LIN {X 0,Y 310.928,Z 762.241,A -85,B 0,C 180,E1 -15746.111,E2 -15746.111} C_VEL
LIN {X 0,Y 310.701,Z 763.849,A -85,B 0,C 180,E1 -15748.703,E2 -15748.703} C_VEL
LIN {X 0,Y 310.698,Z 764.081,A -85,B 0,C 180,E1 -15749.999,E2 -15749.999} C_VEL
LIN {X 0,Y 310.7,Z 763.891,A -85,B 0,C 180,E1 -15751.295,E2 -15751.295} C_VEL
LIN {X 0,Y 310.923,Z 762.339,A -85,B 0,C 180,E1 -15753.887,E2 -15753.887} C_VEL
LIN {X 0,Y 311.084,Z 760.984,A -85,B 0,C 180,E1 -15755.184,E2 -15755.184} C_VEL
LIN {X 0,Y 311.392,Z 758.118,A -85,B 0,C 180,E1 -15757.129,E2 -15757.129} C_VEL
LIN {X 0,Y 311.868,Z 754.229,A -85,B 0,C 180,E1 -15759.075,E2 -15759.075} C_VEL
LIN {X 0,Y 312.703,Z 749.212,A -85,B 0,C 180,E1 -15761.012,E2 -15761.012} C_VEL
LIN {X 0,Y 313.678,Z 742.897,A -85,B 0,C 180,E1 -15762.946,E2 -15762.946} C_VEL
LIN {X 0,Y 314.945,Z 734.989,A -85,B 0,C 180,E1 -15764.868,E2 -15764.868} C_VEL
LIN {X 0,Y 316.624,Z 725.146,A -85,B 0,C 180,E1 -15766.77,E2 -15766.77} C_VEL
LIN {X 0,Y 317.967,Z 714.82,A -85,B 0,C 180,E1 -15768.357,E2 -15768.357} C_VEL
LIN {X 0,Y 319.245,Z 704.591,A -85,B 0,C 180,E1 -15769.615,E2 -15769.615} C_VEL
LIN {X 0,Y 320.576,Z 693.385,A -85,B 0,C 180,E1 -15770.701,E2 -15770.701} C_VEL
LIN {X 0,Y 321.765,Z 680.745,A -85,B 0,C 180,E1 -15771.627,E2 -15771.627} C_VEL
LIN {X 0,Y 322.52,Z 668.996,A -85,B 0,C 180,E1 -15772.247,E2 -15772.247} C_VEL
LIN {X 0,Y 323.102,Z 656.548,A -85,B 0,C 180,E1 -15772.668,E2 -15772.668} C_VEL
LIN {X 0,Y 324.626,Z 584.757,A -85,B 0,C 180,E1 -15774.261,E2 -15774.261} C_VEL
LIN {X 0,Y 322.955,Z 579.324,A -85,B 0,C 180,E1 -15774.526,E2 -15774.526} C_VEL
LIN {X 0,Y 320.223,Z 574.422,A -85,B 0,C 180,E1 -15774.87,E2 -15774.87} C_VEL
LIN {X 0,Y 311.253,Z 562.348,A -85,B 0,C 180,E1 -15775.948,E2 -15775.948} C_VEL
LIN {X 0,Y 309.308,Z 559.08,A -85,B 0,C 180,E1 -15776.208,E2 -15776.208} C_VEL
LIN {X 0,Y 307.194,Z 553.881,A -85,B 0,C 180,E1 -15776.597,E2 -15776.597} C_VEL
LIN {X 0,Y 305.556,Z 546.682,A -85,B 0,C 180,E1 -15779.186,E2 -15779.186} C_VEL
LIN {X 0,Y 305.497,Z 546.411,A -85,B 0,C 180,E1 -15779.66,E2 -15779.66} C_VEL
LIN {X 0,Y 305.462,Z 546.438,A -85,B 0,C 180,E1 -15784.077,E2 -15784.077} C_VEL
LIN {X 0,Y 305.499,Z 546.425,A -85,B 0,C 180,E1 -15786.734,E2 -15786.734} C_VEL
LIN {X 0,Y 305.452,Z 546.427,A -85,B 0,C 180,E1 -15790.599,E2 -15790.599} C_VEL
LIN {X 0,Y 305.423,Z 546.43,A -85,B 0,C 180,E1 -15793.654,E2 -15793.654} C_VEL
LIN {X 0,Y 305.482,Z 546.432,A -85,B 0,C 180,E1 -15797.407,E2 -15797.407} C_VEL
LIN {X 0,Y 305.504,Z 546.404,A -85,B 0,C 180,E1 -15801.601,E2 -15801.601} C_VEL
LIN {X 0,Y 305.458,Z 546.435,A -85,B 0,C 180,E1 -15804.886,E2 -15804.886} C_VEL
LIN {X 0,Y 305.447,Z 546.433,A -85,B 0,C 180,E1 -15808.354,E2 -15808.354} C_VEL
LIN {X 0,Y 305.515,Z 546.426,A -85,B 0,C 180,E1 -15811.113,E2 -15811.113} C_VEL
LIN {X 0,Y 305.565,Z 546.421,A -85,B 0,C 180,E1 -15814.087,E2 -15814.087} C_VEL
LIN {X 0,Y 305.494,Z 546.421,A -85,B 0,C 180,E1 -15818.402,E2 -15818.402} C_VEL
LIN {X 0,Y 305.583,Z 546.42,A -85,B 0,C 180,E1 -15821.217,E2 -15821.217} C_VEL
LIN {X 0,Y 305.642,Z 546.405,A -85,B 0,C 180,E1 -15825.349,E2 -15825.349} C_VEL
LIN {X 0,Y 305.631,Z 546.402,A -85,B 0,C 180,E1 -15829.399,E2 -15829.399} C_VEL
LIN {X 0,Y 305.806,Z 546.391,A -85,B 0,C 180,E1 -15832.074,E2 -15832.074} C_VEL
LIN {X 0,Y 305.683,Z 546.405,A -85,B 0,C 180,E1 -15834.723,E2 -15834.723} C_VEL
LIN {X 0,Y 305.952,Z 546.368,A -85,B 0,C 180,E1 -15838.684,E2 -15838.684} C_VEL
LIN {X 0,Y 305.952,Z 546.374,A -85,B 0,C 180,E1 -15841.316,E2 -15841.316} C_VEL
LIN {X 0,Y 305.847,Z 546.385,A -85,B 0,C 180,E1 -15846.597,E2 -15846.597} C_VEL
LIN {X 0,Y 305.729,Z 546.392,A -85,B 0,C 180,E1 -15849.26,E2 -15849.26} C_VEL
LIN {X 0,Y 305.584,Z 546.42,A -85,B 0,C 180,E1 -15853.296,E2 -15853.296} C_VEL
LIN {X 0,Y 305.587,Z 546.407,A -85,B 0,C 180,E1 -15856.02,E2 -15856.02} C_VEL
LIN {X 0,Y 305.574,Z 546.424,A -85,B 0,C 180,E1 -15859.448,E2 -15859.448} C_VEL
LIN {X 0,Y 305.484,Z 546.427,A -85,B 0,C 180,E1 -15863.042,E2 -15863.042} C_VEL
LIN {X 0,Y 305.519,Z 546.418,A -85,B 0,C 180,E1 -15866.219,E2 -15866.219} C_VEL
LIN {X 0,Y 305.482,Z 546.433,A -85,B 0,C 180,E1 -15869.048,E2 -15869.048} C_VEL
LIN {X 0,Y 305.436,Z 546.436,A -85,B 0,C 180,E1 -15871.953,E2 -15871.953} C_VEL
LIN {X 0,Y 305.457,Z 546.422,A -85,B 0,C 180,E1 -15875.114,E2 -15875.114} C_VEL
LIN {X 0,Y 305.444,Z 546.433,A -85,B 0,C 180,E1 -15878.53,E2 -15878.53} C_VEL
LIN {X 0,Y 305.48,Z 546.416,A -85,B 0,C 180,E1 -15882.593,E2 -15882.593} C_VEL
LIN {X 0,Y 305.488,Z 546.423,A -85,B 0,C 180,E1 -15886.358,E2 -15886.358} C_VEL
LIN {X 0,Y 305.495,Z 546.425,A -85,B 0,C 180,E1 -15889.9,E2 -15889.9} C_VEL
LIN {X 0,Y 305.497,Z 546.41,A -85,B 0,C 180,E1 -15893.628,E2 -15893.628} C_VEL
LIN {X 0,Y 305.507,Z 546.515,A -85,B 0,C 180,E1 -15896.35,E2 -15896.35} C_VEL
LIN {X 0,Y 307.874,Z 556.829,A -85,B 0,C 180,E1 -15899.856,E2 -15899.856} C_VEL
LIN {X 0,Y 309.89,Z 566.829,A -85,B 0,C 180,E1 -15903.028,E2 -15903.028} C_VEL
LIN {X 0,Y 310.333,Z 569.417,A -85,B 0,C 180,E1 -15903.745,E2 -15903.745} C_VEL
LIN {X 0,Y 311.743,Z 574.79,A -85,B 0,C 180,E1 -15904.048,E2 -15904.048} C_VEL
LIN {X 0,Y 316.932,Z 605.166,A -85,B 0,C 180,E1 -15905.243,E2 -15905.243} C_VEL
LIN {X 0,Y 317.713,Z 612.59,A -85,B 0,C 180,E1 -15905.488,E2 -15905.488} C_VEL
LIN {X 0,Y 316.131,Z 677.691,A -85,B 0,C 180,E1 -15906.976,E2 -15906.976} C_VEL
LIN {X 0,Y 315.205,Z 690.854,A -85,B 0,C 180,E1 -15907.511,E2 -15907.511} C_VEL
LIN {X 0,Y 314.128,Z 702.967,A -85,B 0,C 180,E1 -15908.252,E2 -15908.252} C_VEL
LIN {X 0,Y 312.716,Z 715.203,A -85,B 0,C 180,E1 -15909.271,E2 -15909.271} C_VEL
LIN {X 0,Y 311.145,Z 726.778,A -85,B 0,C 180,E1 -15910.54,E2 -15910.54} C_VEL
LIN {X 0,Y 309.567,Z 737.203,A -85,B 0,C 180,E1 -15911.983,E2 -15911.983} C_VEL
LIN {X 0,Y 308.187,Z 746.736,A -85,B 0,C 180,E1 -15913.64,E2 -15913.64} C_VEL
LIN {X 0,Y 306.825,Z 754.98,A -85,B 0,C 180,E1 -15915.408,E2 -15915.408} C_VEL
LIN {X 0,Y 305.546,Z 762.411,A -85,B 0,C 180,E1 -15917.38,E2 -15917.38} C_VEL
LIN {X 0,Y 304.708,Z 768.383,A -85,B 0,C 180,E1 -15919.368,E2 -15919.368} C_VEL
LIN {X 0,Y 304.145,Z 773.106,A -85,B 0,C 180,E1 -15921.363,E2 -15921.363} C_VEL
LIN {X 0,Y 303.739,Z 776.717,A -85,B 0,C 180,E1 -15923.358,E2 -15923.358} C_VEL
LIN {X 0,Y 303.637,Z 778.581,A -85,B 0,C 180,E1 -15924.689,E2 -15924.689} C_VEL
LIN {X 0,Y 303.631,Z 779.979,A -85,B 0,C 180,E1 -15926.019,E2 -15926.019} C_VEL
LIN {X 0,Y 303.607,Z 780.975,A -85,B 0,C 180,E1 -15927.348,E2 -15927.348} C_VEL
LIN {X 0,Y 303.555,Z 781.596,A -85,B 0,C 180,E1 -15928.674,E2 -15928.674} C_VEL
LIN {X 0,Y 303.558,Z 782.931,A -85,B 0,C 180,E1 -15930.001,E2 -15930.001} C_VEL
LIN {X 0,Y 303.543,Z 783.874,A -85,B 0,C 180,E1 -15931.328,E2 -15931.328} C_VEL
LIN {X 0,Y 303.612,Z 784.204,A -85,B 0,C 180,E1 -15932.655,E2 -15932.655} C_VEL
LIN {X 0,Y 303.684,Z 783.949,A -85,B 0,C 180,E1 -15933.982,E2 -15933.982} C_VEL
LIN {X 0,Y 303.863,Z 782.642,A -85,B 0,C 180,E1 -15935.988,E2 -15935.988} C_VEL
LIN {X 0,Y 304.235,Z 780.043,A -85,B 0,C 180,E1 -15937.968,E2 -15937.968} C_VEL
LIN {X 0,Y 304.906,Z 776.069,A -85,B 0,C 180,E1 -15939.956,E2 -15939.956} C_VEL
LIN {X 0,Y 305.765,Z 770.709,A -85,B 0,C 180,E1 -15941.94,E2 -15941.94} C_VEL
LIN {X 0,Y 306.923,Z 763.592,A -85,B 0,C 180,E1 -15943.913,E2 -15943.913} C_VEL
LIN {X 0,Y 308.121,Z 756.001,A -85,B 0,C 180,E1 -15945.547,E2 -15945.547} C_VEL
LIN {X 0,Y 309.196,Z 748.059,A -85,B 0,C 180,E1 -15946.954,E2 -15946.954} C_VEL
LIN {X 0,Y 310.208,Z 738.537,A -85,B 0,C 180,E1 -15948.322,E2 -15948.322} C_VEL
LIN {X 0,Y 311.261,Z 728.283,A -85,B 0,C 180,E1 -15949.455,E2 -15949.455} C_VEL
LIN {X 0,Y 313.548,Z 707.817,A -85,B 0,C 180,E1 -15951.361,E2 -15951.361} C_VEL
LIN {X 0,Y 314.798,Z 695.431,A -85,B 0,C 180,E1 -15952.219,E2 -15952.219} C_VEL
LIN {X 0,Y 315.79,Z 682.684,A -85,B 0,C 180,E1 -15952.836,E2 -15952.836} C_VEL
LIN {X 0,Y 316.351,Z 669.228,A -85,B 0,C 180,E1 -15953.225,E2 -15953.225} C_VEL
LIN {X 0,Y 317.088,Z 640.496,A -85,B 0,C 180,E1 -15953.904,E2 -15953.904} C_VEL
LIN {X 0,Y 319.246,Z 616.116,A -85,B 0,C 180,E1 -15954.917,E2 -15954.917} C_VEL
LIN {X 0,Y 320.405,Z 610.474,A -85,B 0,C 180,E1 -15955.397,E2 -15955.397} C_VEL
LIN {X 0,Y 322.157,Z 595.804,A -85,B 0,C 180,E1 -15957.074,E2 -15957.074} C_VEL
LIN {X 0,Y 322.35,Z 587.346,A -85,B 0,C 180,E1 -15958.391,E2 -15958.391} C_VEL
LIN {X 0,Y 321.375,Z 580.508,A -85,B 0,C 180,E1 -15959.938,E2 -15959.938} C_VEL
LIN {X 0,Y 320.171,Z 573.996,A -85,B 0,C 180,E1 -15961.792,E2 -15961.792} C_VEL
LIN {X 0,Y 319.818,Z 572.14,A -85,B 0,C 180,E1 -15962.423,E2 -15962.423} C_VEL
LIN {X 0,Y 318.873,Z 570.05,A -85,B 0,C 180,E1 -15963.437,E2 -15963.437} C_VEL
LIN {X 0,Y 317.335,Z 567.394,A -85,B 0,C 180,E1 -15965.158,E2 -15965.158} C_VEL
LIN {X 0,Y 316.208,Z 565.397,A -85,B 0,C 180,E1 -15966.878,E2 -15966.878} C_VEL
LIN {X 0,Y 315.21,Z 564.223,A -85,B 0,C 180,E1 -15968.706,E2 -15968.706} C_VEL
LIN {X 0,Y 314.619,Z 563.592,A -85,B 0,C 180,E1 -15970.58,E2 -15970.58} C_VEL
LIN {X 0,Y 314.487,Z 563.578,A -85,B 0,C 180,E1 -15972.484,E2 -15972.484} C_VEL
LIN {X 0,Y 314.722,Z 564.151,A -85,B 0,C 180,E1 -15974.391,E2 -15974.391} C_VEL
LIN {X 0,Y 315.2,Z 565.439,A -85,B 0,C 180,E1 -15976.274,E2 -15976.274} C_VEL
LIN {X 0,Y 316.34,Z 568.507,A -85,B 0,C 180,E1 -15979.058,E2 -15979.058} C_VEL
LIN {X 0,Y 317.765,Z 572.859,A -85,B 0,C 180,E1 -15981.737,E2 -15981.737} C_VEL
LIN {X 0,Y 319.417,Z 578.765,A -85,B 0,C 180,E1 -15984.499,E2 -15984.499} C_VEL
LIN {X 0,Y 320.835,Z 585.947,A -85,B 0,C 180,E1 -15987.161,E2 -15987.161} C_VEL
LIN {X 0,Y 321.558,Z 592.319,A -85,B 0,C 180,E1 -15989.157,E2 -15989.157} C_VEL
LIN {X 0,Y 317.906,Z 611.453,A -85,B 0,C 180,E1 -15993.411,E2 -15993.411} C_VEL
LIN {X 0,Y 316.972,Z 617.933,A -85,B 0,C 180,E1 -15994.77,E2 -15994.77} C_VEL
LIN {X 0,Y 319.921,Z 633.065,A -85,B 0,C 180,E1 -15996.129,E2 -15996.129} C_VEL
LIN {X 0,Y 321.719,Z 645.977,A -85,B 0,C 180,E1 -15997.059,E2 -15997.059} C_VEL
LIN {X 0,Y 321.637,Z 649.738,A -85,B 0,C 180,E1 -15997.236,E2 -15997.236} C_VEL
LIN {X 0,Y 317.807,Z 700.985,A -85,B 0,C 180,E1 -15999.194,E2 -15999.194} C_VEL
LIN {X 0,Y 316.673,Z 711.729,A -85,B 0,C 180,E1 -15999.795,E2 -15999.795} C_VEL
LIN {X 0,Y 315.064,Z 724.183,A -85,B 0,C 180,E1 -16000.791,E2 -16000.791} C_VEL
LIN {X 0,Y 313.669,Z 733.027,A -85,B 0,C 180,E1 -16001.719,E2 -16001.719} C_VEL
LIN {X 0,Y 312.011,Z 742.616,A -85,B 0,C 180,E1 -16002.973,E2 -16002.973} C_VEL
LIN {X 0,Y 310.504,Z 750.378,A -85,B 0,C 180,E1 -16004.24,E2 -16004.24} C_VEL
LIN {X 0,Y 309.197,Z 756.755,A -85,B 0,C 180,E1 -16005.521,E2 -16005.521} C_VEL
LIN {X 0,Y 307.818,Z 763.25,A -85,B 0,C 180,E1 -16007.138,E2 -16007.138} C_VEL
LIN {X 0,Y 306.563,Z 768.489,A -85,B 0,C 180,E1 -16008.763,E2 -16008.763} C_VEL
LIN {X 0,Y 305.426,Z 773.381,A -85,B 0,C 180,E1 -16010.731,E2 -16010.731} C_VEL
LIN {X 0,Y 304.694,Z 776.683,A -85,B 0,C 180,E1 -16012.675,E2 -16012.675} C_VEL
LIN {X 0,Y 304.123,Z 778.808,A -85,B 0,C 180,E1 -16014.696,E2 -16014.696} C_VEL
LIN {X 0,Y 303.833,Z 779.547,A -85,B 0,C 180,E1 -16016.021,E2 -16016.021} C_VEL
LIN {X 0,Y 303.656,Z 779.771,A -85,B 0,C 180,E1 -16017.347,E2 -16017.347} C_VEL
LIN {X 0,Y 303.549,Z 779.408,A -85,B 0,C 180,E1 -16018.673,E2 -16018.673} C_VEL
LIN {X 0,Y 303.534,Z 778.447,A -85,B 0,C 180,E1 -16020,E2 -16020} C_VEL
LIN {X 0,Y 303.566,Z 776.051,A -85,B 0,C 180,E1 -16021.99,E2 -16021.99} C_VEL
LIN {X 0,Y 303.8,Z 772.192,A -85,B 0,C 180,E1 -16023.98,E2 -16023.98} C_VEL
LIN {X 0,Y 303.878,Z 766.731,A -85,B 0,C 180,E1 -16026.011,E2 -16026.011} C_VEL
LIN {X 0,Y 304.292,Z 759.714,A -85,B 0,C 180,E1 -16027.966,E2 -16027.966} C_VEL
LIN {X 0,Y 304.608,Z 753.688,A -85,B 0,C 180,E1 -16029.294,E2 -16029.294} C_VEL
LIN {X 0,Y 305.115,Z 745.403,A -85,B 0,C 180,E1 -16030.787,E2 -16030.787} C_VEL
LIN {X 0,Y 305.671,Z 736.328,A -85,B 0,C 180,E1 -16032.111,E2 -16032.111} C_VEL
LIN {X 0,Y 306.288,Z 726.07,A -85,B 0,C 180,E1 -16033.265,E2 -16033.265} C_VEL
LIN {X 0,Y 306.799,Z 716.759,A -85,B 0,C 180,E1 -16034.087,E2 -16034.087} C_VEL
LIN {X 0,Y 307.116,Z 707.091,A -85,B 0,C 180,E1 -16034.749,E2 -16034.749} C_VEL
LIN {X 0,Y 307.563,Z 695.072,A -85,B 0,C 180,E1 -16035.32,E2 -16035.32} C_VEL
LIN {X 0,Y 308.869,Z 641.052,A -85,B 0,C 180,E1 -16037.122,E2 -16037.122} C_VEL
LIN {X 0,Y 306.94,Z 618.294,A -85,B 0,C 180,E1 -16037.963,E2 -16037.963} C_VEL
LIN {X 0,Y 306.926,Z 616.972,A -85,B 0,C 180,E1 -16038.05,E2 -16038.05} C_VEL
LIN {X 0,Y 308.497,Z 593.246,A -85,B 0,C 180,E1 -16042.786,E2 -16042.786} C_VEL
LIN {X 0,Y 309.943,Z 574.161,A -85,B 0,C 180,E1 -16046.605,E2 -16046.605} C_VEL
LIN {X 0,Y 310.246,Z 569.759,A -85,B 0,C 180,E1 -16047.495,E2 -16047.495} C_VEL
LIN {X 0,Y 308.04,Z 558.66,A -85,B 0,C 180,E1 -16049.889,E2 -16049.889} C_VEL
LIN {X 0,Y 305.53,Z 546.557,A -85,B 0,C 180,E1 -16052.6,E2 -16052.6} C_VEL
LIN {X 0,Y 305.501,Z 546.43,A -85,B 0,C 180,E1 -16056.736,E2 -16056.736} C_VEL
LIN {X 0,Y 305.458,Z 546.398,A -85,B 0,C 180,E1 -16060.599,E2 -16060.599} C_VEL
LIN {X 0,Y 305.429,Z 546.397,A -85,B 0,C 180,E1 -16063.655,E2 -16063.655} C_VEL
LIN {X 0,Y 305.459,Z 546.432,A -85,B 0,C 180,E1 -16067.414,E2 -16067.414} C_VEL
LIN {X 0,Y 305.471,Z 546.407,A -85,B 0,C 180,E1 -16071.596,E2 -16071.596} C_VEL
LIN {X 0,Y 305.466,Z 546.425,A -85,B 0,C 180,E1 -16074.886,E2 -16074.886} C_VEL
LIN {X 0,Y 305.453,Z 546.43,A -85,B 0,C 180,E1 -16078.355,E2 -16078.355} C_VEL
LIN {X 0,Y 305.528,Z 546.479,A -85,B 0,C 180,E1 -16080.805,E2 -16080.805} C_VEL
LIN {X 0,Y 307.121,Z 553.574,A -85,B 0,C 180,E1 -16083.444,E2 -16083.444} C_VEL
LIN {X 0,Y 307.557,Z 555.027,A -85,B 0,C 180,E1 -16083.632,E2 -16083.632} C_VEL
LIN {X 0,Y 314.364,Z 571.517,A -85,B 0,C 180,E1 -16084.671,E2 -16084.671} C_VEL
LIN {X 0,Y 316.455,Z 577.198,A -85,B 0,C 180,E1 -16084.992,E2 -16084.992} C_VEL
LIN {X 0,Y 318.23,Z 587.126,A -85,B 0,C 180,E1 -16085.385,E2 -16085.385} C_VEL
LIN {X 0,Y 316.331,Z 660.198,A -85,B 0,C 180,E1 -16087.033,E2 -16087.033} C_VEL
LIN {X 0,Y 315.671,Z 673.592,A -85,B 0,C 180,E1 -16087.587,E2 -16087.587} C_VEL
LIN {X 0,Y 314.802,Z 685.224,A -85,B 0,C 180,E1 -16088.298,E2 -16088.298} C_VEL
LIN {X 0,Y 313.447,Z 697.673,A -85,B 0,C 180,E1 -16089.319,E2 -16089.319} C_VEL
LIN {X 0,Y 311.953,Z 709.318,A -85,B 0,C 180,E1 -16090.59,E2 -16090.59} C_VEL
LIN {X 0,Y 310.582,Z 719.633,A -85,B 0,C 180,E1 -16092.02,E2 -16092.02} C_VEL
LIN {X 0,Y 309.279,Z 728.306,A -85,B 0,C 180,E1 -16093.497,E2 -16093.497} C_VEL
LIN {X 0,Y 307.94,Z 736.173,A -85,B 0,C 180,E1 -16095.121,E2 -16095.121} C_VEL
LIN {X 0,Y 306.641,Z 743.857,A -85,B 0,C 180,E1 -16097.086,E2 -16097.086} C_VEL
LIN {X 0,Y 305.411,Z 750.913,A -85,B 0,C 180,E1 -16099.391,E2 -16099.391} C_VEL
LIN {X 0,Y 304.678,Z 755.609,A -85,B 0,C 180,E1 -16101.376,E2 -16101.376} C_VEL
LIN {X 0,Y 304.196,Z 759.318,A -85,B 0,C 180,E1 -16103.442,E2 -16103.442} C_VEL
LIN {X 0,Y 304.024,Z 761.05,A -85,B 0,C 180,E1 -16104.693,E2 -16104.693} C_VEL
LIN {X 0,Y 303.867,Z 762.446,A -85,B 0,C 180,E1 -16106.02,E2 -16106.02} C_VEL
LIN {X 0,Y 303.617,Z 764.054,A -85,B 0,C 180,E1 -16108.672,E2 -16108.672} C_VEL
LIN {X 0,Y 303.611,Z 764.285,A -85,B 0,C 180,E1 -16109.999,E2 -16109.999} C_VEL
LIN {X 0,Y 303.617,Z 764.095,A -85,B 0,C 180,E1 -16111.325,E2 -16111.325} C_VEL
LIN {X 0,Y 303.862,Z 762.543,A -85,B 0,C 180,E1 -16113.978,E2 -16113.978} C_VEL
LIN {X 0,Y 304.019,Z 761.188,A -85,B 0,C 180,E1 -16115.304,E2 -16115.304} C_VEL
LIN {X 0,Y 304.345,Z 758.321,A -85,B 0,C 180,E1 -16117.295,E2 -16117.295} C_VEL
LIN {X 0,Y 304.844,Z 754.433,A -85,B 0,C 180,E1 -16119.286,E2 -16119.286} C_VEL
LIN {X 0,Y 305.715,Z 749.416,A -85,B 0,C 180,E1 -16121.267,E2 -16121.267} C_VEL
LIN {X 0,Y 306.746,Z 743.101,A -85,B 0,C 180,E1 -16123.244,E2 -16123.244} C_VEL
LIN {X 0,Y 308.104,Z 735.19,A -85,B 0,C 180,E1 -16125.207,E2 -16125.207} C_VEL
LIN {X 0,Y 309.826,Z 725.348,A -85,B 0,C 180,E1 -16127.15,E2 -16127.15} C_VEL
LIN {X 0,Y 311.235,Z 715.02,A -85,B 0,C 180,E1 -16128.769,E2 -16128.769} C_VEL
LIN {X 0,Y 312.565,Z 704.791,A -85,B 0,C 180,E1 -16130.052,E2 -16130.052} C_VEL
LIN {X 0,Y 313.962,Z 693.583,A -85,B 0,C 180,E1 -16131.158,E2 -16131.158} C_VEL
LIN {X 0,Y 315.177,Z 680.941,A -85,B 0,C 180,E1 -16132.103,E2 -16132.103} C_VEL
LIN {X 0,Y 316.065,Z 668.273,A -85,B 0,C 180,E1 -16132.769,E2 -16132.769} C_VEL
LIN {X 0,Y 316.594,Z 655.229,A -85,B 0,C 180,E1 -16133.204,E2 -16133.204} C_VEL
LIN {X 0,Y 318.197,Z 585.811,A -85,B 0,C 180,E1 -16134.763,E2 -16134.763} C_VEL
LIN {X 0,Y 315.996,Z 575.74,A -85,B 0,C 180,E1 -16135.197,E2 -16135.197} C_VEL
LIN {X 0,Y 309.308,Z 559.08,A -85,B 0,C 180,E1 -16136.208,E2 -16136.208} C_VEL
LIN {X 0,Y 307.198,Z 556.188,A -85,B 0,C 180,E1 -16136.544,E2 -16136.544} C_VEL
LIN {X 0,Y 303.944,Z 553.527,A -85,B 0,C 180,E1 -16137.187,E2 -16137.187} C_VEL
LIN {X 0,Y 300.339,Z 551.127,A -85,B 0,C 180,E1 -16138.211,E2 -16138.211} C_VEL
LIN {X 0,Y 298.896,Z 549.304,A -85,B 0,C 180,E1 -16139.018,E2 -16139.018} C_VEL
LIN {X 0,Y 298.807,Z 549.001,A -85,B 0,C 180,E1 -16139.136,E2 -16139.136} C_VEL
LIN {X 0,Y 298.451,Z 547.324,A -85,B 0,C 180,E1 -16139.879,E2 -16139.879} C_VEL
LIN {X 0,Y 298.425,Z 547.314,A -85,B 0,C 180,E1 -16144.486,E2 -16144.486} C_VEL
LIN {X 0,Y 298.434,Z 547.313,A -85,B 0,C 180,E1 -16147.753,E2 -16147.753} C_VEL
LIN {X 0,Y 298.382,Z 547.313,A -85,B 0,C 180,E1 -16151.26,E2 -16151.26} C_VEL
LIN {X 0,Y 298.35,Z 547.302,A -85,B 0,C 180,E1 -16155.034,E2 -16155.034} C_VEL
LIN {X 0,Y 298.427,Z 547.307,A -85,B 0,C 180,E1 -16156.925,E2 -16156.925} C_VEL
LIN {X 0,Y 298.421,Z 547.286,A -85,B 0,C 180,E1 -16161,E2 -16161} C_VEL
LIN {X 0,Y 298.428,Z 547.307,A -85,B 0,C 180,E1 -16163.931,E2 -16163.931} C_VEL
LIN {X 0,Y 298.39,Z 547.31,A -85,B 0,C 180,E1 -16167.982,E2 -16167.982} C_VEL
LIN {X 0,Y 298.458,Z 547.297,A -85,B 0,C 180,E1 -16171.904,E2 -16171.904} C_VEL
LIN {X 0,Y 298.479,Z 547.304,A -85,B 0,C 180,E1 -16174.923,E2 -16174.923} C_VEL
LIN {X 0,Y 298.443,Z 547.303,A -85,B 0,C 180,E1 -16179.315,E2 -16179.315} C_VEL
LIN {X 0,Y 298.531,Z 547.292,A -85,B 0,C 180,E1 -16182.179,E2 -16182.179} C_VEL
LIN {X 0,Y 298.586,Z 547.281,A -85,B 0,C 180,E1 -16184.994,E2 -16184.994} C_VEL
LIN {X 0,Y 298.586,Z 547.281,A -85,B 0,C 180,E1 -16189.146,E2 -16189.146} C_VEL
LIN {X 0,Y 298.751,Z 547.266,A -85,B 0,C 180,E1 -16191.886,E2 -16191.886} C_VEL
LIN {X 0,Y 298.654,Z 547.28,A -85,B 0,C 180,E1 -16194.599,E2 -16194.599} C_VEL
LIN {X 0,Y 298.918,Z 547.244,A -85,B 0,C 180,E1 -16198.653,E2 -16198.653} C_VEL
LIN {X 0,Y 298.918,Z 547.249,A -85,B 0,C 180,E1 -16201.347,E2 -16201.347} C_VEL
LIN {X 0,Y 298.792,Z 547.264,A -85,B 0,C 180,E1 -16206.754,E2 -16206.754} C_VEL
LIN {X 0,Y 298.673,Z 547.268,A -85,B 0,C 180,E1 -16209.481,E2 -16209.481} C_VEL
LIN {X 0,Y 298.546,Z 547.297,A -85,B 0,C 180,E1 -16213.616,E2 -16213.616} C_VEL
LIN {X 0,Y 298.542,Z 547.285,A -85,B 0,C 180,E1 -16216.409,E2 -16216.409} C_VEL
LIN {X 0,Y 298.509,Z 547.301,A -85,B 0,C 180,E1 -16219.658,E2 -16219.658} C_VEL
LIN {X 0,Y 298.451,Z 547.308,A -85,B 0,C 180,E1 -16223.598,E2 -16223.598} C_VEL
LIN {X 0,Y 298.477,Z 547.295,A -85,B 0,C 180,E1 -16226.576,E2 -16226.576} C_VEL
LIN {X 0,Y 298.41,Z 547.313,A -85,B 0,C 180,E1 -16229.642,E2 -16229.642} C_VEL
LIN {X 0,Y 298.389,Z 547.315,A -85,B 0,C 180,E1 -16232.801,E2 -16232.801} C_VEL
LIN {X 0,Y 298.441,Z 547.284,A -85,B 0,C 180,E1 -16236.809,E2 -16236.809} C_VEL
LIN {X 0,Y 298.409,Z 547.305,A -85,B 0,C 180,E1 -16241.258,E2 -16241.258} C_VEL
LIN {X 0,Y 298.412,Z 547.314,A -85,B 0,C 180,E1 -16245.048,E2 -16245.048} C_VEL
LIN {X 0,Y 298.45,Z 547.309,A -85,B 0,C 180,E1 -16248.751,E2 -16248.751} C_VEL
LIN {X 0,Y 298.463,Z 547.279,A -85,B 0,C 180,E1 -16253.188,E2 -16253.188} C_VEL
LIN {X 0,Y 298.426,Z 547.398,A -85,B 0,C 180,E1 -16255.789,E2 -16255.789} C_VEL
LIN {X 0,Y 300.554,Z 556.606,A -85,B 0,C 180,E1 -16259.042,E2 -16259.042} C_VEL
LIN {X 0,Y 302.687,Z 566.604,A -85,B 0,C 180,E1 -16262.332,E2 -16262.332} C_VEL
LIN {X 0,Y 303.15,Z 569.151,A -85,B 0,C 180,E1 -16263.067,E2 -16263.067} C_VEL
LIN {X 0,Y 305.199,Z 575.223,A -85,B 0,C 180,E1 -16263.464,E2 -16263.464} C_VEL
LIN {X 0,Y 310.189,Z 604.178,A -85,B 0,C 180,E1 -16264.648,E2 -16264.648} C_VEL
LIN {X 0,Y 311.274,Z 613.377,A -85,B 0,C 180,E1 -16264.971,E2 -16264.971} C_VEL
LIN {X 0,Y 309.619,Z 677.5,A -85,B 0,C 180,E1 -16266.463,E2 -16266.463} C_VEL
LIN {X 0,Y 308.592,Z 691.42,A -85,B 0,C 180,E1 -16267.046,E2 -16267.046} C_VEL
LIN {X 0,Y 307.436,Z 703.883,A -85,B 0,C 180,E1 -16267.842,E2 -16267.842} C_VEL
LIN {X 0,Y 306.079,Z 715.003,A -85,B 0,C 180,E1 -16268.8,E2 -16268.8} C_VEL
LIN {X 0,Y 304.434,Z 726.577,A -85,B 0,C 180,E1 -16270.093,E2 -16270.093} C_VEL
LIN {X 0,Y 302.795,Z 737,A -85,B 0,C 180,E1 -16271.566,E2 -16271.566} C_VEL
LIN {X 0,Y 301.509,Z 745.549,A -85,B 0,C 180,E1 -16273.065,E2 -16273.065} C_VEL
LIN {X 0,Y 300.188,Z 753.4,A -85,B 0,C 180,E1 -16274.73,E2 -16274.73} C_VEL
LIN {X 0,Y 298.808,Z 761.086,A -85,B 0,C 180,E1 -16276.744,E2 -16276.744} C_VEL
LIN {X 0,Y 297.712,Z 768.179,A -85,B 0,C 180,E1 -16279.115,E2 -16279.115} C_VEL
LIN {X 0,Y 297.087,Z 772.901,A -85,B 0,C 180,E1 -16281.156,E2 -16281.156} C_VEL
LIN {X 0,Y 296.686,Z 776.513,A -85,B 0,C 180,E1 -16283.199,E2 -16283.199} C_VEL
LIN {X 0,Y 296.552,Z 778.376,A -85,B 0,C 180,E1 -16284.562,E2 -16284.562} C_VEL
LIN {X 0,Y 296.528,Z 779.774,A -85,B 0,C 180,E1 -16285.924,E2 -16285.924} C_VEL
LIN {X 0,Y 296.533,Z 780.771,A -85,B 0,C 180,E1 -16287.284,E2 -16287.284} C_VEL
LIN {X 0,Y 296.476,Z 781.38,A -85,B 0,C 180,E1 -16288.643,E2 -16288.643} C_VEL
LIN {X 0,Y 296.465,Z 783.647,A -85,B 0,C 180,E1 -16291.36,E2 -16291.36} C_VEL
LIN {X 0,Y 296.54,Z 784.068,A -85,B 0,C 180,E1 -16292.718,E2 -16292.718} C_VEL
LIN {X 0,Y 296.585,Z 783.961,A -85,B 0,C 180,E1 -16294.078,E2 -16294.078} C_VEL
LIN {X 0,Y 296.748,Z 782.985,A -85,B 0,C 180,E1 -16295.898,E2 -16295.898} C_VEL
LIN {X 0,Y 296.863,Z 782.201,A -85,B 0,C 180,E1 -16296.799,E2 -16296.799} C_VEL
LIN {X 0,Y 297.418,Z 779.335,A -85,B 0,C 180,E1 -16298.836,E2 -16298.836} C_VEL
LIN {X 0,Y 298.219,Z 775.165,A -85,B 0,C 180,E1 -16300.868,E2 -16300.868} C_VEL
LIN {X 0,Y 299.232,Z 769.575,A -85,B 0,C 180,E1 -16302.894,E2 -16302.894} C_VEL
LIN {X 0,Y 300.414,Z 763.501,A -85,B 0,C 180,E1 -16304.567,E2 -16304.567} C_VEL
LIN {X 0,Y 301.455,Z 757.619,A -85,B 0,C 180,E1 -16305.9,E2 -16305.9} C_VEL
LIN {X 0,Y 302.652,Z 749.943,A -85,B 0,C 180,E1 -16307.332,E2 -16307.332} C_VEL
LIN {X 0,Y 303.808,Z 741.089,A -85,B 0,C 180,E1 -16308.711,E2 -16308.711} C_VEL
LIN {X 0,Y 305.137,Z 730.156,A -85,B 0,C 180,E1 -16310.037,E2 -16310.037} C_VEL
LIN {X 0,Y 306.125,Z 719.612,A -85,B 0,C 180,E1 -16311.022,E2 -16311.022} C_VEL
LIN {X 0,Y 306.931,Z 708.781,A -85,B 0,C 180,E1 -16311.801,E2 -16311.801} C_VEL
LIN {X 0,Y 308.476,Z 692.512,A -85,B 0,C 180,E1 -16312.877,E2 -16312.877} C_VEL
LIN {X 0,Y 309.506,Z 679.117,A -85,B 0,C 180,E1 -16313.46,E2 -16313.46} C_VEL
LIN {X 0,Y 310.162,Z 660.267,A -85,B 0,C 180,E1 -16313.983,E2 -16313.983} C_VEL
LIN {X 0,Y 314.234,Z 616.296,A -85,B 0,C 180,E1 -16315.834,E2 -16315.834} C_VEL
LIN {X 0,Y 315.071,Z 612.858,A -85,B 0,C 180,E1 -16316.128,E2 -16316.128} C_VEL
LIN {X 0,Y 317.004,Z 599.024,A -85,B 0,C 180,E1 -16317.748,E2 -16317.748} C_VEL
LIN {X 0,Y 317.391,Z 591.84,A -85,B 0,C 180,E1 -16318.876,E2 -16318.876} C_VEL
LIN {X 0,Y 316.852,Z 586.233,A -85,B 0,C 180,E1 -16320.112,E2 -16320.112} C_VEL
LIN {X 0,Y 315.603,Z 578.659,A -85,B 0,C 180,E1 -16322.307,E2 -16322.307} C_VEL
LIN {X 0,Y 315.162,Z 576.897,A -85,B 0,C 180,E1 -16322.962,E2 -16322.962} C_VEL
LIN {X 0,Y 313.468,Z 573.781,A -85,B 0,C 180,E1 -16324.8,E2 -16324.8} C_VEL
LIN {X 0,Y 312.589,Z 572.232,A -85,B 0,C 180,E1 -16325.963,E2 -16325.963} C_VEL
LIN {X 0,Y 311.445,Z 570.49,A -85,B 0,C 180,E1 -16327.833,E2 -16327.833} C_VEL
LIN {X 0,Y 310.584,Z 569.514,A -85,B 0,C 180,E1 -16329.703,E2 -16329.703} C_VEL
LIN {X 0,Y 310.131,Z 569.243,A -85,B 0,C 180,E1 -16332.832,E2 -16332.832} C_VEL
LIN {X 0,Y 310.457,Z 570.272,A -85,B 0,C 180,E1 -16335.431,E2 -16335.431} C_VEL
LIN {X 0,Y 311.264,Z 572.748,A -85,B 0,C 180,E1 -16338.169,E2 -16338.169} C_VEL
LIN {X 0,Y 312.44,Z 576.747,A -85,B 0,C 180,E1 -16340.962,E2 -16340.962} C_VEL
LIN {X 0,Y 313.853,Z 582.097,A -85,B 0,C 180,E1 -16343.721,E2 -16343.721} C_VEL
LIN {X 0,Y 314.977,Z 587.939,A -85,B 0,C 180,E1 -16346.095,E2 -16346.095} C_VEL
LIN {X 0,Y 315.813,Z 595.108,A -85,B 0,C 180,E1 -16348.532,E2 -16348.532} C_VEL
LIN {X 0,Y 315.065,Z 599.161,A -85,B 0,C 180,E1 -16349.504,E2 -16349.504} C_VEL
LIN {X 0,Y 311.39,Z 617.879,A -85,B 0,C 180,E1 -16353.695,E2 -16353.695} C_VEL
LIN {X 0,Y 314.189,Z 632.181,A -85,B 0,C 180,E1 -16355.081,E2 -16355.081} C_VEL
LIN {X 0,Y 316.047,Z 645.065,A -85,B 0,C 180,E1 -16356.122,E2 -16356.122} C_VEL
LIN {X 0,Y 316.296,Z 649.045,A -85,B 0,C 180,E1 -16356.381,E2 -16356.381} C_VEL
LIN {X 0,Y 312.13,Z 700.711,A -85,B 0,C 180,E1 -16358.408,E2 -16358.408} C_VEL
LIN {X 0,Y 310.844,Z 711.935,A -85,B 0,C 180,E1 -16359.053,E2 -16359.053} C_VEL
LIN {X 0,Y 309.134,Z 724.263,A -85,B 0,C 180,E1 -16360.061,E2 -16360.061} C_VEL
LIN {X 0,Y 307.634,Z 733.129,A -85,B 0,C 180,E1 -16361.001,E2 -16361.001} C_VEL
LIN {X 0,Y 305.873,Z 742.706,A -85,B 0,C 180,E1 -16362.275,E2 -16362.275} C_VEL
LIN {X 0,Y 303.829,Z 752.039,A -85,B 0,C 180,E1 -16363.884,E2 -16363.884} C_VEL
LIN {X 0,Y 302.466,Z 758.11,A -85,B 0,C 180,E1 -16365.191,E2 -16365.191} C_VEL
LIN {X 0,Y 301.008,Z 764.416,A -85,B 0,C 180,E1 -16366.842,E2 -16366.842} C_VEL
LIN {X 0,Y 299.675,Z 769.478,A -85,B 0,C 180,E1 -16368.502,E2 -16368.502} C_VEL
LIN {X 0,Y 298.448,Z 774.034,A -85,B 0,C 180,E1 -16370.512,E2 -16370.512} C_VEL
LIN {X 0,Y 297.872,Z 776.32,A -85,B 0,C 180,E1 -16371.862,E2 -16371.862} C_VEL
LIN {X 0,Y 297.458,Z 777.984,A -85,B 0,C 180,E1 -16373.216,E2 -16373.216} C_VEL
LIN {X 0,Y 297.07,Z 779.095,A -85,B 0,C 180,E1 -16374.57,E2 -16374.57} C_VEL
LIN {X 0,Y 296.76,Z 779.685,A -85,B 0,C 180,E1 -16375.926,E2 -16375.926} C_VEL
LIN {X 0,Y 296.587,Z 779.76,A -85,B 0,C 180,E1 -16377.284,E2 -16377.284} C_VEL
LIN {X 0,Y 296.471,Z 779.313,A -85,B 0,C 180,E1 -16378.642,E2 -16378.642} C_VEL
LIN {X 0,Y 296.452,Z 778.281,A -85,B 0,C 180,E1 -16380,E2 -16380} C_VEL
LIN {X 0,Y 296.493,Z 775.638,A -85,B 0,C 180,E1 -16382.038,E2 -16382.038} C_VEL
LIN {X 0,Y 296.649,Z 773.167,A -85,B 0,C 180,E1 -16383.396,E2 -16383.396} C_VEL
LIN {X 0,Y 296.69,Z 769.984,A -85,B 0,C 180,E1 -16384.756,E2 -16384.756} C_VEL
LIN {X 0,Y 297.006,Z 763.754,A -85,B 0,C 180,E1 -16386.795,E2 -16386.795} C_VEL
LIN {X 0,Y 297.253,Z 758.552,A -85,B 0,C 180,E1 -16388.156,E2 -16388.156} C_VEL
LIN {X 0,Y 297.576,Z 752.283,A -85,B 0,C 180,E1 -16389.516,E2 -16389.516} C_VEL
LIN {X 0,Y 298.135,Z 743.721,A -85,B 0,C 180,E1 -16391.042,E2 -16391.042} C_VEL
LIN {X 0,Y 298.731,Z 734.012,A -85,B 0,C 180,E1 -16392.397,E2 -16392.397} C_VEL
LIN {X 0,Y 299.272,Z 724.898,A -85,B 0,C 180,E1 -16393.409,E2 -16393.409} C_VEL
LIN {X 0,Y 299.891,Z 713.261,A -85,B 0,C 180,E1 -16394.418,E2 -16394.418} C_VEL
LIN {X 0,Y 300.189,Z 702.017,A -85,B 0,C 180,E1 -16395.097,E2 -16395.097} C_VEL
LIN {X 0,Y 300.725,Z 688.753,A -85,B 0,C 180,E1 -16395.634,E2 -16395.634} C_VEL
LIN {X 0,Y 301.689,Z 639.978,A -85,B 0,C 180,E1 -16397.335,E2 -16397.335} C_VEL
LIN {X 0,Y 299.899,Z 618.487,A -85,B 0,C 180,E1 -16398.134,E2 -16398.134} C_VEL
LIN {X 0,Y 299.878,Z 616.836,A -85,B 0,C 180,E1 -16398.268,E2 -16398.268} C_VEL
LIN {X 0,Y 301.37,Z 595.335,A -85,B 0,C 180,E1 -16402.63,E2 -16402.63} C_VEL
LIN {X 0,Y 302.866,Z 576.151,A -85,B 0,C 180,E1 -16406.532,E2 -16406.532} C_VEL
LIN {X 0,Y 303.253,Z 570.852,A -85,B 0,C 180,E1 -16407.614,E2 -16407.614} C_VEL
LIN {X 0,Y 300.878,Z 559.082,A -85,B 0,C 180,E1 -16410.2,E2 -16410.2} C_VEL
LIN {X 0,Y 298.487,Z 547.424,A -85,B 0,C 180,E1 -16412.864,E2 -16412.864} C_VEL
LIN {X 0,Y 298.469,Z 547.306,A -85,B 0,C 180,E1 -16416.812,E2 -16416.812} C_VEL
LIN {X 0,Y 298.39,Z 547.269,A -85,B 0,C 180,E1 -16421.087,E2 -16421.087} C_VEL
LIN {X 0,Y 298.403,Z 547.264,A -85,B 0,C 180,E1 -16423.103,E2 -16423.103} C_VEL
LIN {X 0,Y 298.407,Z 547.316,A -85,B 0,C 180,E1 -16426.92,E2 -16426.92} C_VEL
LIN {X 0,Y 298.402,Z 547.28,A -85,B 0,C 180,E1 -16431.007,E2 -16431.007} C_VEL
LIN {X 0,Y 298.422,Z 547.312,A -85,B 0,C 180,E1 -16433.93,E2 -16433.93} C_VEL
LIN {X 0,Y 298.397,Z 547.312,A -85,B 0,C 180,E1 -16437.983,E2 -16437.983} C_VEL
LIN {X 0,Y 298.48,Z 547.466,A -85,B 0,C 180,E1 -16440.364,E2 -16440.364} C_VEL
LIN {X 0,Y 300.019,Z 554.107,A -85,B 0,C 180,E1 -16442.831,E2 -16442.831} C_VEL
LIN {X 0,Y 302.341,Z 559.588,A -85,B 0,C 180,E1 -16443.266,E2 -16443.266} C_VEL
LIN {X 0,Y 309.544,Z 577.444,A -85,B 0,C 180,E1 -16444.394,E2 -16444.394} C_VEL
LIN {X 0,Y 310.639,Z 581.388,A -85,B 0,C 180,E1 -16444.591,E2 -16444.591} C_VEL
LIN {X 0,Y 311.778,Z 588.206,A -85,B 0,C 180,E1 -16444.861,E2 -16444.861} C_VEL
LIN {X 0,Y 309.901,Z 658.988,A -85,B 0,C 180,E1 -16446.484,E2 -16446.484} C_VEL
LIN {X 0,Y 309.373,Z 671.51,A -85,B 0,C 180,E1 -16446.972,E2 -16446.972} C_VEL
LIN {X 0,Y 308.316,Z 684.309,A -85,B 0,C 180,E1 -16447.729,E2 -16447.729} C_VEL
LIN {X 0,Y 307.041,Z 696.146,A -85,B 0,C 180,E1 -16448.692,E2 -16448.692} C_VEL
LIN {X 0,Y 305.672,Z 706.893,A -85,B 0,C 180,E1 -16449.825,E2 -16449.825} C_VEL
LIN {X 0,Y 304.255,Z 716.776,A -85,B 0,C 180,E1 -16451.131,E2 -16451.131} C_VEL
LIN {X 0,Y 302.803,Z 726.739,A -85,B 0,C 180,E1 -16452.786,E2 -16452.786} C_VEL
LIN {X 0,Y 301.066,Z 736.381,A -85,B 0,C 180,E1 -16454.774,E2 -16454.774} C_VEL
LIN {X 0,Y 299.724,Z 744.064,A -85,B 0,C 180,E1 -16456.783,E2 -16456.783} C_VEL
LIN {X 0,Y 298.438,Z 751.119,A -85,B 0,C 180,E1 -16459.14,E2 -16459.14} C_VEL
LIN {X 0,Y 297.638,Z 755.816,A -85,B 0,C 180,E1 -16461.17,E2 -16461.17} C_VEL
LIN {X 0,Y 297.119,Z 759.774,A -85,B 0,C 180,E1 -16463.447,E2 -16463.447} C_VEL
LIN {X 0,Y 296.785,Z 762.651,A -85,B 0,C 180,E1 -16465.925,E2 -16465.925} C_VEL
LIN {X 0,Y 296.536,Z 764.258,A -85,B 0,C 180,E1 -16468.641,E2 -16468.641} C_VEL
LIN {X 0,Y 296.526,Z 764.49,A -85,B 0,C 180,E1 -16469.999,E2 -16469.999} C_VEL
LIN {X 0,Y 296.535,Z 764.299,A -85,B 0,C 180,E1 -16471.357,E2 -16471.357} C_VEL
LIN {X 0,Y 296.78,Z 762.747,A -85,B 0,C 180,E1 -16474.073,E2 -16474.073} C_VEL
LIN {X 0,Y 297.09,Z 760.011,A -85,B 0,C 180,E1 -16476.504,E2 -16476.504} C_VEL
LIN {X 0,Y 297.635,Z 756.05,A -85,B 0,C 180,E1 -16478.828,E2 -16478.828} C_VEL
LIN {X 0,Y 298.411,Z 751.418,A -85,B 0,C 180,E1 -16480.859,E2 -16480.859} C_VEL
LIN {X 0,Y 299.656,Z 744.434,A -85,B 0,C 180,E1 -16483.218,E2 -16483.218} C_VEL
LIN {X 0,Y 300.977,Z 736.862,A -85,B 0,C 180,E1 -16485.229,E2 -16485.229} C_VEL
LIN {X 0,Y 302.769,Z 727.325,A -85,B 0,C 180,E1 -16487.214,E2 -16487.214} C_VEL
LIN {X 0,Y 304.202,Z 717.485,A -85,B 0,C 180,E1 -16488.87,E2 -16488.87} C_VEL
LIN {X 0,Y 305.548,Z 707.802,A -85,B 0,C 180,E1 -16490.182,E2 -16490.182} C_VEL
LIN {X 0,Y 306.93,Z 697.308,A -85,B 0,C 180,E1 -16491.314,E2 -16491.314} C_VEL
LIN {X 0,Y 308.346,Z 684.655,A -85,B 0,C 180,E1 -16492.354,E2 -16492.354} C_VEL
LIN {X 0,Y 309.302,Z 671.992,A -85,B 0,C 180,E1 -16493.119,E2 -16493.119} C_VEL
LIN {X 0,Y 309.898,Z 659.917,A -85,B 0,C 180,E1 -16493.603,E2 -16493.603} C_VEL
LIN {X 0,Y 311.28,Z 609.925,A -85,B 0,C 180,E1 -16494.754,E2 -16494.754} C_VEL
LIN {X 0,Y 311.745,Z 587.035,A -85,B 0,C 180,E1 -16495.285,E2 -16495.285} C_VEL
LIN {X 0,Y 309.882,Z 578.32,A -85,B 0,C 180,E1 -16495.669,E2 -16495.669} C_VEL
LIN {X 0,Y 302.493,Z 560.002,A -85,B 0,C 180,E1 -16496.826,E2 -16496.826} C_VEL
LIN {X 0,Y 300.076,Z 554.221,A -85,B 0,C 180,E1 -16497.262,E2 -16497.262} C_VEL
LIN {X 0,Y 298.807,Z 549.001,A -85,B 0,C 180,E1 -16499.136,E2 -16499.136} C_VEL
LIN {X 0,Y 298.156,Z 547.825,A -85,B 0,C 180,E1 -16499.823,E2 -16499.823} C_VEL
LIN {X 0,Y 297.152,Z 547.457,A -85,B 0,C 180,E1 -16500.538,E2 -16500.538} C_VEL
LIN {X 0,Y 292.405,Z 548.127,A -85,B 0,C 180,E1 -16503.519,E2 -16503.519} C_VEL
LIN {X 0,Y 291.46,Z 548.186,A -85,B 0,C 180,E1 -16504.697,E2 -16504.697} C_VEL
LIN {X 0,Y 291.383,Z 548.185,A -85,B 0,C 180,E1 -16505.095,E2 -16505.095} C_VEL
LIN {X 0,Y 291.396,Z 548.185,A -85,B 0,C 180,E1 -16507.259,E2 -16507.259} C_VEL
LIN {X 0,Y 291.332,Z 548.186,A -85,B 0,C 180,E1 -16510.641,E2 -16510.641} C_VEL
LIN {X 0,Y 291.285,Z 548.183,A -85,B 0,C 180,E1 -16514.401,E2 -16514.401} C_VEL
LIN {X 0,Y 291.351,Z 548.192,A -85,B 0,C 180,E1 -16518.397,E2 -16518.397} C_VEL
LIN {X 0,Y 291.37,Z 548.163,A -85,B 0,C 180,E1 -16521.161,E2 -16521.161} C_VEL
LIN {X 0,Y 291.381,Z 548.188,A -85,B 0,C 180,E1 -16524.629,E2 -16524.629} C_VEL
LIN {X 0,Y 291.367,Z 548.185,A -85,B 0,C 180,E1 -16527.95,E2 -16527.95} C_VEL
LIN {X 0,Y 291.377,Z 548.186,A -85,B 0,C 180,E1 -16531.158,E2 -16531.158} C_VEL
LIN {X 0,Y 291.411,Z 548.184,A -85,B 0,C 180,E1 -16534.271,E2 -16534.271} C_VEL
LIN {X 0,Y 291.375,Z 548.179,A -85,B 0,C 180,E1 -16537.299,E2 -16537.299} C_VEL
LIN {X 0,Y 291.451,Z 548.178,A -85,B 0,C 180,E1 -16540.27,E2 -16540.27} C_VEL
LIN {X 0,Y 291.548,Z 548.157,A -85,B 0,C 180,E1 -16544.623,E2 -16544.623} C_VEL
LIN {X 0,Y 291.53,Z 548.163,A -85,B 0,C 180,E1 -16548.88,E2 -16548.88} C_VEL
LIN {X 0,Y 291.702,Z 548.141,A -85,B 0,C 180,E1 -16551.688,E2 -16551.688} C_VEL
LIN {X 0,Y 291.625,Z 548.156,A -85,B 0,C 180,E1 -16554.468,E2 -16554.468} C_VEL
LIN {X 0,Y 291.884,Z 548.12,A -85,B 0,C 180,E1 -16558.62,E2 -16558.62} C_VEL
LIN {X 0,Y 291.884,Z 548.125,A -85,B 0,C 180,E1 -16561.38,E2 -16561.38} C_VEL
LIN {X 0,Y 291.74,Z 548.143,A -85,B 0,C 180,E1 -16566.918,E2 -16566.918} C_VEL
LIN {X 0,Y 291.622,Z 548.145,A -85,B 0,C 180,E1 -16569.712,E2 -16569.712} C_VEL
LIN {X 0,Y 291.516,Z 548.17,A -85,B 0,C 180,E1 -16573.951,E2 -16573.951} C_VEL
LIN {X 0,Y 291.48,Z 548.165,A -85,B 0,C 180,E1 -16576.818,E2 -16576.818} C_VEL
LIN {X 0,Y 291.444,Z 548.179,A -85,B 0,C 180,E1 -16579.875,E2 -16579.875} C_VEL
LIN {X 0,Y 291.393,Z 548.188,A -85,B 0,C 180,E1 -16584.206,E2 -16584.206} C_VEL
LIN {X 0,Y 291.408,Z 548.177,A -85,B 0,C 180,E1 -16587.273,E2 -16587.273} C_VEL
LIN {X 0,Y 291.328,Z 548.19,A -85,B 0,C 180,E1 -16590.438,E2 -16590.438} C_VEL
LIN {X 0,Y 291.339,Z 548.193,A -85,B 0,C 180,E1 -16593.699,E2 -16593.699} C_VEL
LIN {X 0,Y 291.37,Z 548.167,A -85,B 0,C 180,E1 -16597.255,E2 -16597.255} C_VEL
LIN {X 0,Y 291.365,Z 548.189,A -85,B 0,C 180,E1 -16600.637,E2 -16600.637} C_VEL
LIN {X 0,Y 291.338,Z 548.195,A -85,B 0,C 180,E1 -16604.393,E2 -16604.393} C_VEL
LIN {X 0,Y 291.384,Z 548.187,A -85,B 0,C 180,E1 -16608.392,E2 -16608.392} C_VEL
LIN {X 0,Y 291.378,Z 548.16,A -85,B 0,C 180,E1 -16611.164,E2 -16611.164} C_VEL
LIN {X 0,Y 291.382,Z 548.187,A -85,B 0,C 180,E1 -16614.631,E2 -16614.631} C_VEL
LIN {X 0,Y 291.396,Z 548.295,A -85,B 0,C 180,E1 -16615.219,E2 -16615.219} C_VEL
LIN {X 0,Y 293.507,Z 557.422,A -85,B 0,C 180,E1 -16618.547,E2 -16618.547} C_VEL
LIN {X 0,Y 295.723,Z 567.833,A -85,B 0,C 180,E1 -16622.07,E2 -16622.07} C_VEL
LIN {X 0,Y 295.98,Z 569.047,A -85,B 0,C 180,E1 -16622.373,E2 -16622.373} C_VEL
LIN {X 0,Y 299.033,Z 577.373,A -85,B 0,C 180,E1 -16622.934,E2 -16622.934} C_VEL
LIN {X 0,Y 303.917,Z 605.992,A -85,B 0,C 180,E1 -16624.137,E2 -16624.137} C_VEL
LIN {X 0,Y 304.849,Z 614.165,A -85,B 0,C 180,E1 -16624.431,E2 -16624.431} C_VEL
LIN {X 0,Y 303.13,Z 677.308,A -85,B 0,C 180,E1 -16625.928,E2 -16625.928} C_VEL
LIN {X 0,Y 302.126,Z 690.462,A -85,B 0,C 180,E1 -16626.48,E2 -16626.48} C_VEL
LIN {X 0,Y 301,Z 702.571,A -85,B 0,C 180,E1 -16627.251,E2 -16627.251} C_VEL
LIN {X 0,Y 299.479,Z 714.803,A -85,B 0,C 180,E1 -16628.31,E2 -16628.31} C_VEL
LIN {X 0,Y 297.765,Z 726.376,A -85,B 0,C 180,E1 -16629.628,E2 -16629.628} C_VEL
LIN {X 0,Y 296.054,Z 736.798,A -85,B 0,C 180,E1 -16631.13,E2 -16631.13} C_VEL
LIN {X 0,Y 294.579,Z 746.053,A -85,B 0,C 180,E1 -16632.801,E2 -16632.801} C_VEL
LIN {X 0,Y 293.036,Z 754.572,A -85,B 0,C 180,E1 -16634.705,E2 -16634.705} C_VEL
LIN {X 0,Y 291.654,Z 762.004,A -85,B 0,C 180,E1 -16636.768,E2 -16636.768} C_VEL
LIN {X 0,Y 290.722,Z 767.975,A -85,B 0,C 180,E1 -16638.85,E2 -16638.85} C_VEL
LIN {X 0,Y 290.048,Z 772.696,A -85,B 0,C 180,E1 -16640.94,E2 -16640.94} C_VEL
LIN {X 0,Y 289.607,Z 776.309,A -85,B 0,C 180,E1 -16643.032,E2 -16643.032} C_VEL
LIN {X 0,Y 289.478,Z 778.259,A -85,B 0,C 180,E1 -16644.507,E2 -16644.507} C_VEL
LIN {X 0,Y 289.438,Z 780.567,A -85,B 0,C 180,E1 -16647.218,E2 -16647.218} C_VEL
LIN {X 0,Y 289.398,Z 781.173,A -85,B 0,C 180,E1 -16648.61,E2 -16648.61} C_VEL
LIN {X 0,Y 289.389,Z 783.36,A -85,B 0,C 180,E1 -16651.393,E2 -16651.393} C_VEL
LIN {X 0,Y 289.448,Z 783.928,A -85,B 0,C 180,E1 -16652.785,E2 -16652.785} C_VEL
LIN {X 0,Y 289.491,Z 783.98,A -85,B 0,C 180,E1 -16654.178,E2 -16654.178} C_VEL
LIN {X 0,Y 289.675,Z 783.288,A -85,B 0,C 180,E1 -16655.884,E2 -16655.884} C_VEL
LIN {X 0,Y 289.816,Z 782.475,A -85,B 0,C 180,E1 -16656.965,E2 -16656.965} C_VEL
LIN {X 0,Y 290.428,Z 779.841,A -85,B 0,C 180,E1 -16659.051,E2 -16659.051} C_VEL
LIN {X 0,Y 291.279,Z 775.887,A -85,B 0,C 180,E1 -16661.13,E2 -16661.13} C_VEL
LIN {X 0,Y 292.389,Z 770.552,A -85,B 0,C 180,E1 -16663.201,E2 -16663.201} C_VEL
LIN {X 0,Y 293.94,Z 763.468,A -85,B 0,C 180,E1 -16665.25,E2 -16665.25} C_VEL
LIN {X 0,Y 295.397,Z 756.007,A -85,B 0,C 180,E1 -16666.944,E2 -16666.944} C_VEL
LIN {X 0,Y 296.71,Z 748.245,A -85,B 0,C 180,E1 -16668.39,E2 -16668.39} C_VEL
LIN {X 0,Y 298.117,Z 738.81,A -85,B 0,C 180,E1 -16669.81,E2 -16669.81} C_VEL
LIN {X 0,Y 299.419,Z 728.963,A -85,B 0,C 180,E1 -16670.975,E2 -16670.975} C_VEL
LIN {X 0,Y 300.57,Z 718.432,A -85,B 0,C 180,E1 -16671.971,E2 -16671.971} C_VEL
LIN {X 0,Y 301.55,Z 706.525,A -85,B 0,C 180,E1 -16672.798,E2 -16672.798} C_VEL
LIN {X 0,Y 302.625,Z 687.227,A -85,B 0,C 180,E1 -16673.753,E2 -16673.753} C_VEL
LIN {X 0,Y 309.417,Z 616.568,A -85,B 0,C 180,E1 -16676.795,E2 -16676.795} C_VEL
LIN {X 0,Y 310.127,Z 613.106,A -85,B 0,C 180,E1 -16677.135,E2 -16677.135} C_VEL
LIN {X 0,Y 312.03,Z 601.541,A -85,B 0,C 180,E1 -16678.548,E2 -16678.548} C_VEL
LIN {X 0,Y 312.47,Z 594.845,A -85,B 0,C 180,E1 -16679.659,E2 -16679.659} C_VEL
LIN {X 0,Y 311.855,Z 588.987,A -85,B 0,C 180,E1 -16681.088,E2 -16681.088} C_VEL
LIN {X 0,Y 311.004,Z 583.312,A -85,B 0,C 180,E1 -16682.845,E2 -16682.845} C_VEL
LIN {X 0,Y 310.162,Z 581.12,A -85,B 0,C 180,E1 -16683.879,E2 -16683.879} C_VEL
LIN {X 0,Y 308.143,Z 577.589,A -85,B 0,C 180,E1 -16686.371,E2 -16686.371} C_VEL
LIN {X 0,Y 306.723,Z 575.628,A -85,B 0,C 180,E1 -16688.826,E2 -16688.826} C_VEL
LIN {X 0,Y 306.056,Z 574.944,A -85,B 0,C 180,E1 -16690.731,E2 -16690.731} C_VEL
LIN {X 0,Y 305.75,Z 574.998,A -85,B 0,C 180,E1 -16693.598,E2 -16693.598} C_VEL
LIN {X 0,Y 305.983,Z 575.786,A -85,B 0,C 180,E1 -16695.401,E2 -16695.401} C_VEL
LIN {X 0,Y 306.672,Z 578.403,A -85,B 0,C 180,E1 -16698.349,E2 -16698.349} C_VEL
LIN {X 0,Y 307.616,Z 582.085,A -85,B 0,C 180,E1 -16700.968,E2 -16700.968} C_VEL
LIN {X 0,Y 308.77,Z 587.303,A -85,B 0,C 180,E1 -16703.715,E2 -16703.715} C_VEL
LIN {X 0,Y 309.57,Z 592.144,A -85,B 0,C 180,E1 -16705.764,E2 -16705.764} C_VEL
LIN {X 0,Y 310.169,Z 597.954,A -85,B 0,C 180,E1 -16707.846,E2 -16707.846} C_VEL
LIN {X 0,Y 309.822,Z 600.572,A -85,B 0,C 180,E1 -16708.551,E2 -16708.551} C_VEL
LIN {X 0,Y 306.084,Z 617.81,A -85,B 0,C 180,E1 -16712.524,E2 -16712.524} C_VEL
LIN {X 0,Y 308.608,Z 631.32,A -85,B 0,C 180,E1 -16713.96,E2 -16713.96} C_VEL
LIN {X 0,Y 310.621,Z 645.195,A -85,B 0,C 180,E1 -16715.177,E2 -16715.177} C_VEL
LIN {X 0,Y 310.97,Z 650.777,A -85,B 0,C 180,E1 -16715.557,E2 -16715.557} C_VEL
LIN {X 0,Y 306.466,Z 701.614,A -85,B 0,C 180,E1 -16717.633,E2 -16717.633} C_VEL
LIN {X 0,Y 304.955,Z 713.802,A -85,B 0,C 180,E1 -16718.362,E2 -16718.362} C_VEL
LIN {X 0,Y 303.304,Z 724.685,A -85,B 0,C 180,E1 -16719.307,E2 -16719.307} C_VEL
LIN {X 0,Y 301.712,Z 733.385,A -85,B 0,C 180,E1 -16720.26,E2 -16720.26} C_VEL
LIN {X 0,Y 299.739,Z 742.851,A -85,B 0,C 180,E1 -16721.546,E2 -16721.546} C_VEL
LIN {X 0,Y 297.577,Z 752.177,A -85,B 0,C 180,E1 -16723.183,E2 -16723.183} C_VEL
LIN {X 0,Y 296.09,Z 758.258,A -85,B 0,C 180,E1 -16724.512,E2 -16724.512} C_VEL
LIN {X 0,Y 294.825,Z 763.342,A -85,B 0,C 180,E1 -16725.857,E2 -16725.857} C_VEL
LIN {X 0,Y 293.302,Z 768.568,A -85,B 0,C 180,E1 -16727.546,E2 -16727.546} C_VEL
LIN {X 0,Y 291.874,Z 773.461,A -85,B 0,C 180,E1 -16729.596,E2 -16729.596} C_VEL
LIN {X 0,Y 290.87,Z 776.822,A -85,B 0,C 180,E1 -16731.664,E2 -16731.664} C_VEL
LIN {X 0,Y 290.414,Z 778.409,A -85,B 0,C 180,E1 -16733.05,E2 -16733.05} C_VEL
LIN {X 0,Y 290.02,Z 779.395,A -85,B 0,C 180,E1 -16734.438,E2 -16734.438} C_VEL
LIN {X 0,Y 289.689,Z 779.824,A -85,B 0,C 180,E1 -16735.826,E2 -16735.826} C_VEL
LIN {X 0,Y 289.498,Z 779.744,A -85,B 0,C 180,E1 -16737.217,E2 -16737.217} C_VEL
LIN {X 0,Y 289.395,Z 779.147,A -85,B 0,C 180,E1 -16738.608,E2 -16738.608} C_VEL
LIN {X 0,Y 289.373,Z 778.018,A -85,B 0,C 180,E1 -16740,E2 -16740} C_VEL
LIN {X 0,Y 289.423,Z 775.14,A -85,B 0,C 180,E1 -16742.087,E2 -16742.087} C_VEL
LIN {X 0,Y 289.624,Z 770.936,A -85,B 0,C 180,E1 -16744.175,E2 -16744.175} C_VEL
LIN {X 0,Y 289.714,Z 766.134,A -85,B 0,C 180,E1 -16745.954,E2 -16745.954} C_VEL
LIN {X 0,Y 290.09,Z 760.249,A -85,B 0,C 180,E1 -16747.657,E2 -16747.657} C_VEL
LIN {X 0,Y 290.359,Z 754.289,A -85,B 0,C 180,E1 -16749.052,E2 -16749.052} C_VEL
LIN {X 0,Y 290.848,Z 746.06,A -85,B 0,C 180,E1 -16750.617,E2 -16750.617} C_VEL
LIN {X 0,Y 291.466,Z 737.097,A -85,B 0,C 180,E1 -16752.004,E2 -16752.004} C_VEL
LIN {X 0,Y 292.052,Z 727.091,A -85,B 0,C 180,E1 -16753.215,E2 -16753.215} C_VEL
LIN {X 0,Y 292.606,Z 717.015,A -85,B 0,C 180,E1 -16754.164,E2 -16754.164} C_VEL
LIN {X 0,Y 292.952,Z 707.503,A -85,B 0,C 180,E1 -16754.856,E2 -16754.856} C_VEL
LIN {X 0,Y 293.423,Z 694.838,A -85,B 0,C 180,E1 -16755.499,E2 -16755.499} C_VEL
LIN {X 0,Y 294.761,Z 641.997,A -85,B 0,C 180,E1 -16757.404,E2 -16757.404} C_VEL
LIN {X 0,Y 292.858,Z 618.593,A -85,B 0,C 180,E1 -16758.314,E2 -16758.314} C_VEL
LIN {X 0,Y 292.84,Z 616.875,A -85,B 0,C 180,E1 -16758.451,E2 -16758.451} C_VEL
LIN {X 0,Y 294.233,Z 597.401,A -85,B 0,C 180,E1 -16762.469,E2 -16762.469} C_VEL
LIN {X 0,Y 295.789,Z 578.102,A -85,B 0,C 180,E1 -16766.456,E2 -16766.456} C_VEL
LIN {X 0,Y 296.205,Z 572.779,A -85,B 0,C 180,E1 -16767.56,E2 -16767.56} C_VEL
LIN {X 0,Y 295.386,Z 567.104,A -85,B 0,C 180,E1 -16768.802,E2 -16768.802} C_VEL
LIN {X 0,Y 291.443,Z 548.358,A -85,B 0,C 180,E1 -16773.087,E2 -16773.087} C_VEL
LIN {X 0,Y 291.399,Z 548.189,A -85,B 0,C 180,E1 -16777.258,E2 -16777.258} C_VEL
LIN {X 0,Y 291.338,Z 548.153,A -85,B 0,C 180,E1 -16780.642,E2 -16780.642} C_VEL
LIN {X 0,Y 291.294,Z 548.169,A -85,B 0,C 180,E1 -16784.402,E2 -16784.402} C_VEL
LIN {X 0,Y 291.33,Z 548.176,A -85,B 0,C 180,E1 -16788.404,E2 -16788.404} C_VEL
LIN {X 0,Y 291.351,Z 548.159,A -85,B 0,C 180,E1 -16791.157,E2 -16791.157} C_VEL
LIN {X 0,Y 291.365,Z 548.183,A -85,B 0,C 180,E1 -16794.625,E2 -16794.625} C_VEL
LIN {X 0,Y 291.374,Z 548.186,A -85,B 0,C 180,E1 -16797.95,E2 -16797.95} C_VEL
LIN {X 0,Y 291.402,Z 548.289,A -85,B 0,C 180,E1 -16799.771,E2 -16799.771} C_VEL
LIN {X 0,Y 292.814,Z 554.338,A -85,B 0,C 180,E1 -16802.106,E2 -16802.106} C_VEL
LIN {X 0,Y 295.4,Z 560.275,A -85,B 0,C 180,E1 -16802.597,E2 -16802.597} C_VEL
LIN {X 0,Y 302.449,Z 577.321,A -85,B 0,C 180,E1 -16803.738,E2 -16803.738} C_VEL
LIN {X 0,Y 304.393,Z 583.29,A -85,B 0,C 180,E1 -16804.074,E2 -16804.074} C_VEL
LIN {X 0,Y 305.379,Z 588.434,A -85,B 0,C 180,E1 -16804.297,E2 -16804.297} C_VEL
LIN {X 0,Y 303.422,Z 659.213,A -85,B 0,C 180,E1 -16805.95,E2 -16805.95} C_VEL
LIN {X 0,Y 302.864,Z 671.726,A -85,B 0,C 180,E1 -16806.448,E2 -16806.448} C_VEL
LIN {X 0,Y 301.756,Z 684.522,A -85,B 0,C 180,E1 -16807.218,E2 -16807.218} C_VEL
LIN {X 0,Y 300.457,Z 696.356,A -85,B 0,C 180,E1 -16808.201,E2 -16808.201} C_VEL
LIN {X 0,Y 299.009,Z 707.103,A -85,B 0,C 180,E1 -16809.355,E2 -16809.355} C_VEL
LIN {X 0,Y 297.549,Z 716.984,A -85,B 0,C 180,E1 -16810.689,E2 -16810.689} C_VEL
LIN {X 0,Y 296.025,Z 726.946,A -85,B 0,C 180,E1 -16812.379,E2 -16812.379} C_VEL
LIN {X 0,Y 294.222,Z 736.588,A -85,B 0,C 180,E1 -16814.41,E2 -16814.41} C_VEL
LIN {X 0,Y 292.812,Z 744.271,A -85,B 0,C 180,E1 -16816.465,E2 -16816.465} C_VEL
LIN {X 0,Y 291.474,Z 751.325,A -85,B 0,C 180,E1 -16818.877,E2 -16818.877} C_VEL
LIN {X 0,Y 290.624,Z 756.022,A -85,B 0,C 180,E1 -16820.955,E2 -16820.955} C_VEL
LIN {X 0,Y 290.035,Z 760.229,A -85,B 0,C 180,E1 -16823.463,E2 -16823.463} C_VEL
LIN {X 0,Y 289.706,Z 762.856,A -85,B 0,C 180,E1 -16825.825,E2 -16825.825} C_VEL
LIN {X 0,Y 289.457,Z 764.463,A -85,B 0,C 180,E1 -16828.608,E2 -16828.608} C_VEL
LIN {X 0,Y 289.444,Z 764.694,A -85,B 0,C 180,E1 -16829.999,E2 -16829.999} C_VEL
LIN {X 0,Y 289.457,Z 764.503,A -85,B 0,C 180,E1 -16831.39,E2 -16831.39} C_VEL
LIN {X 0,Y 289.701,Z 762.951,A -85,B 0,C 180,E1 -16834.172,E2 -16834.172} C_VEL
LIN {X 0,Y 290.014,Z 760.422,A -85,B 0,C 180,E1 -16836.501,E2 -16836.501} C_VEL
LIN {X 0,Y 290.62,Z 756.253,A -85,B 0,C 180,E1 -16839.042,E2 -16839.042} C_VEL
LIN {X 0,Y 291.443,Z 751.621,A -85,B 0,C 180,E1 -16841.122,E2 -16841.122} C_VEL
LIN {X 0,Y 292.717,Z 744.638,A -85,B 0,C 180,E1 -16843.537,E2 -16843.537} C_VEL
LIN {X 0,Y 294.146,Z 737.064,A -85,B 0,C 180,E1 -16845.591,E2 -16845.591} C_VEL
LIN {X 0,Y 295.999,Z 727.527,A -85,B 0,C 180,E1 -16847.62,E2 -16847.62} C_VEL
LIN {X 0,Y 297.481,Z 717.687,A -85,B 0,C 180,E1 -16849.313,E2 -16849.313} C_VEL
LIN {X 0,Y 298.917,Z 708.001,A -85,B 0,C 180,E1 -16850.65,E2 -16850.65} C_VEL
LIN {X 0,Y 300.35,Z 697.506,A -85,B 0,C 180,E1 -16851.805,E2 -16851.805} C_VEL
LIN {X 0,Y 301.8,Z 684.851,A -85,B 0,C 180,E1 -16852.866,E2 -16852.866} C_VEL
LIN {X 0,Y 302.804,Z 672.186,A -85,B 0,C 180,E1 -16853.645,E2 -16853.645} C_VEL
LIN {X 0,Y 303.423,Z 660.101,A -85,B 0,C 180,E1 -16854.138,E2 -16854.138} C_VEL
LIN {X 0,Y 304.996,Z 603.749,A -85,B 0,C 180,E1 -16855.462,E2 -16855.462} C_VEL
LIN {X 0,Y 305.247,Z 587.572,A -85,B 0,C 180,E1 -16855.853,E2 -16855.853} C_VEL
LIN {X 0,Y 303.672,Z 580.476,A -85,B 0,C 180,E1 -16856.182,E2 -16856.182} C_VEL
LIN {X 0,Y 296.337,Z 562.402,A -85,B 0,C 180,E1 -16857.37,E2 -16857.37} C_VEL
LIN {X 0,Y 292.832,Z 554.451,A -85,B 0,C 180,E1 -16857.994,E2 -16857.994} C_VEL
LIN {X 0,Y 291.441,Z 548.492,A -85,B 0,C 180,E1 -16860.225,E2 -16860.225} C_VEL
LIN {X 0,Y 291.384,Z 548.208,A -85,B 0,C 180,E1 -16860.43,E2 -16860.43} C_VEL
LIN {X 0,Y 291.387,Z 548.187,A -85,B 0,C 180,E1 -16864.91,E2 -16864.91} C_VEL
LIN {X 0,Y 291.383,Z 548.185,A -85,B 0,C 180,E1 -16865.095,E2 -16865.095} C_VEL
LIN {X 0,Y 290.702,Z 548.267,A -85,B 0,C 180,E1 -16866.247,E2 -16866.247} C_VEL
LIN {X 0,Y 287.81,Z 548.634,A -85,B 0,C 180,E1 -16868.122,E2 -16868.122} C_VEL
LIN {X 0,Y 285.365,Z 548.93,A -85,B 0,C 180,E1 -16869.645,E2 -16869.645} C_VEL
LIN {X 0,Y 284.326,Z 549.06,A -85,B 0,C 180,E1 -16870.826,E2 -16870.826} C_VEL
LIN {X 0,Y 284.246,Z 549.071,A -85,B 0,C 180,E1 -16871.226,E2 -16871.226} C_VEL
LIN {X 0,Y 284.241,Z 549.062,A -85,B 0,C 180,E1 -16874.189,E2 -16874.189} C_VEL
LIN {X 0,Y 284.298,Z 549.071,A -85,B 0,C 180,E1 -16878.129,E2 -16878.129} C_VEL
LIN {X 0,Y 284.325,Z 549.041,A -85,B 0,C 180,E1 -16881.833,E2 -16881.833} C_VEL
LIN {X 0,Y 284.319,Z 549.072,A -85,B 0,C 180,E1 -16885.352,E2 -16885.352} C_VEL
LIN {X 0,Y 284.29,Z 549.068,A -85,B 0,C 180,E1 -16888.725,E2 -16888.725} C_VEL
LIN {X 0,Y 284.391,Z 549.048,A -85,B 0,C 180,E1 -16892.825,E2 -16892.825} C_VEL
LIN {X 0,Y 284.36,Z 549.058,A -85,B 0,C 180,E1 -16896.706,E2 -16896.706} C_VEL
LIN {X 0,Y 284.398,Z 549.06,A -85,B 0,C 180,E1 -16901.261,E2 -16901.261} C_VEL
LIN {X 0,Y 284.485,Z 549.036,A -85,B 0,C 180,E1 -16904.459,E2 -16904.459} C_VEL
LIN {X 0,Y 284.481,Z 549.042,A -85,B 0,C 180,E1 -16908.601,E2 -16908.601} C_VEL
LIN {X 0,Y 284.652,Z 549.017,A -85,B 0,C 180,E1 -16911.481,E2 -16911.481} C_VEL
LIN {X 0,Y 284.595,Z 549.032,A -85,B 0,C 180,E1 -16914.331,E2 -16914.331} C_VEL
LIN {X 0,Y 284.85,Z 548.997,A -85,B 0,C 180,E1 -16918.586,E2 -16918.586} C_VEL
LIN {X 0,Y 284.85,Z 549,A -85,B 0,C 180,E1 -16921.414,E2 -16921.414} C_VEL
LIN {X 0,Y 284.692,Z 549.022,A -85,B 0,C 180,E1 -16927.09,E2 -16927.09} C_VEL
LIN {X 0,Y 284.56,Z 549.023,A -85,B 0,C 180,E1 -16929.956,E2 -16929.956} C_VEL
LIN {X 0,Y 284.475,Z 549.045,A -85,B 0,C 180,E1 -16934.303,E2 -16934.303} C_VEL
LIN {X 0,Y 284.419,Z 549.047,A -85,B 0,C 180,E1 -16937.249,E2 -16937.249} C_VEL
LIN {X 0,Y 284.372,Z 549.058,A -85,B 0,C 180,E1 -16940.243,E2 -16940.243} C_VEL
LIN {X 0,Y 284.363,Z 549.066,A -85,B 0,C 180,E1 -16943.876,E2 -16943.876} C_VEL
LIN {X 0,Y 284.385,Z 549.051,A -85,B 0,C 180,E1 -16947.172,E2 -16947.172} C_VEL
LIN {X 0,Y 284.288,Z 549.066,A -85,B 0,C 180,E1 -16951.275,E2 -16951.275} C_VEL
LIN {X 0,Y 284.335,Z 549.048,A -85,B 0,C 180,E1 -16955.349,E2 -16955.349} C_VEL
LIN {X 0,Y 284.307,Z 549.057,A -85,B 0,C 180,E1 -16958.17,E2 -16958.17} C_VEL
LIN {X 0,Y 284.292,Z 549.055,A -85,B 0,C 180,E1 -16962.132,E2 -16962.132} C_VEL
LIN {X 0,Y 284.313,Z 549.061,A -85,B 0,C 180,E1 -16966.203,E2 -16966.203} C_VEL
LIN {X 0,Y 284.347,Z 549.055,A -85,B 0,C 180,E1 -16970.014,E2 -16970.014} C_VEL
LIN {X 0,Y 284.336,Z 549.053,A -85,B 0,C 180,E1 -16974.197,E2 -16974.197} C_VEL
LIN {X 0,Y 284.373,Z 549.32,A -85,B 0,C 180,E1 -16974.713,E2 -16974.713} C_VEL
LIN {X 0,Y 286.568,Z 558.667,A -85,B 0,C 180,E1 -16978.181,E2 -16978.181} C_VEL
LIN {X 0,Y 288.658,Z 568.548,A -85,B 0,C 180,E1 -16981.573,E2 -16981.573} C_VEL
LIN {X 0,Y 290.758,Z 574.019,A -85,B 0,C 180,E1 -16982.013,E2 -16982.013} C_VEL
LIN {X 0,Y 292.982,Z 579.883,A -85,B 0,C 180,E1 -16982.401,E2 -16982.401} C_VEL
LIN {X 0,Y 297.797,Z 608.866,A -85,B 0,C 180,E1 -16983.645,E2 -16983.645} C_VEL
LIN {X 0,Y 298.442,Z 615.511,A -85,B 0,C 180,E1 -16983.881,E2 -16983.881} C_VEL
LIN {X 0,Y 296.674,Z 677.117,A -85,B 0,C 180,E1 -16985.37,E2 -16985.37} C_VEL
LIN {X 0,Y 295.576,Z 691.029,A -85,B 0,C 180,E1 -16985.973,E2 -16985.973} C_VEL
LIN {X 0,Y 294.332,Z 703.486,A -85,B 0,C 180,E1 -16986.799,E2 -16986.799} C_VEL
LIN {X 0,Y 292.889,Z 714.603,A -85,B 0,C 180,E1 -16987.796,E2 -16987.796} C_VEL
LIN {X 0,Y 291.098,Z 726.174,A -85,B 0,C 180,E1 -16989.14,E2 -16989.14} C_VEL
LIN {X 0,Y 289.324,Z 736.596,A -85,B 0,C 180,E1 -16990.674,E2 -16990.674} C_VEL
LIN {X 0,Y 287.878,Z 744.947,A -85,B 0,C 180,E1 -16992.197,E2 -16992.197} C_VEL
LIN {X 0,Y 286.405,Z 752.992,A -85,B 0,C 180,E1 -16993.976,E2 -16993.976} C_VEL
LIN {X 0,Y 284.968,Z 760.679,A -85,B 0,C 180,E1 -16996.088,E2 -16996.088} C_VEL
LIN {X 0,Y 284.001,Z 765.948,A -85,B 0,C 180,E1 -16997.859,E2 -16997.859} C_VEL
LIN {X 0,Y 283.2,Z 771.056,A -85,B 0,C 180,E1 -16999.997,E2 -16999.997} C_VEL
LIN {X 0,Y 282.684,Z 775.03,A -85,B 0,C 180,E1 -17002.142,E2 -17002.142} C_VEL
LIN {X 0,Y 282.37,Z 778.301,A -85,B 0,C 180,E1 -17004.609,E2 -17004.609} C_VEL
LIN {X 0,Y 282.345,Z 780.362,A -85,B 0,C 180,E1 -17007.148,E2 -17007.148} C_VEL
LIN {X 0,Y 282.316,Z 781.811,A -85,B 0,C 180,E1 -17010.001,E2 -17010.001} C_VEL
LIN {X 0,Y 282.314,Z 783.043,A -85,B 0,C 180,E1 -17011.428,E2 -17011.428} C_VEL
LIN {X 0,Y 282.358,Z 783.781,A -85,B 0,C 180,E1 -17012.855,E2 -17012.855} C_VEL
LIN {X 0,Y 282.402,Z 784,A -85,B 0,C 180,E1 -17014.283,E2 -17014.283} C_VEL
LIN {X 0,Y 282.595,Z 783.569,A -85,B 0,C 180,E1 -17015.855,E2 -17015.855} C_VEL
LIN {X 0,Y 282.763,Z 782.674,A -85,B 0,C 180,E1 -17017.14,E2 -17017.14} C_VEL
LIN {X 0,Y 283.161,Z 781.212,A -85,B 0,C 180,E1 -17018.565,E2 -17018.565} C_VEL
LIN {X 0,Y 284.05,Z 778.01,A -85,B 0,C 180,E1 -17020.695,E2 -17020.695} C_VEL
LIN {X 0,Y 285.154,Z 773.451,A -85,B 0,C 180,E1 -17022.817,E2 -17022.817} C_VEL
LIN {X 0,Y 286.368,Z 768.449,A -85,B 0,C 180,E1 -17024.571,E2 -17024.571} C_VEL
LIN {X 0,Y 287.856,Z 762.202,A -85,B 0,C 180,E1 -17026.307,E2 -17026.307} C_VEL
LIN {X 0,Y 289.143,Z 756.16,A -85,B 0,C 180,E1 -17027.689,E2 -17027.689} C_VEL
LIN {X 0,Y 290.901,Z 747.084,A -85,B 0,C 180,E1 -17029.404,E2 -17029.404} C_VEL
LIN {X 0,Y 292.427,Z 737.998,A -85,B 0,C 180,E1 -17030.763,E2 -17030.763} C_VEL
LIN {X 0,Y 293.862,Z 728.048,A -85,B 0,C 180,E1 -17031.944,E2 -17031.944} C_VEL
LIN {X 0,Y 295.394,Z 715.305,A -85,B 0,C 180,E1 -17033.115,E2 -17033.115} C_VEL
LIN {X 0,Y 296.41,Z 703.194,A -85,B 0,C 180,E1 -17033.911,E2 -17033.911} C_VEL
LIN {X 0,Y 298.031,Z 681.048,A -85,B 0,C 180,E1 -17034.978,E2 -17034.978} C_VEL
LIN {X 0,Y 304.785,Z 616.911,A -85,B 0,C 180,E1 -17037.797,E2 -17037.797} C_VEL
LIN {X 0,Y 307.232,Z 603.565,A -85,B 0,C 180,E1 -17039.462,E2 -17039.462} C_VEL
LIN {X 0,Y 307.624,Z 598.254,A -85,B 0,C 180,E1 -17040.412,E2 -17040.412} C_VEL
LIN {X 0,Y 307.118,Z 593.048,A -85,B 0,C 180,E1 -17041.759,E2 -17041.759} C_VEL
LIN {X 0,Y 306.445,Z 587.989,A -85,B 0,C 180,E1 -17043.397,E2 -17043.397} C_VEL
LIN {X 0,Y 304.926,Z 584.922,A -85,B 0,C 180,E1 -17045.185,E2 -17045.185} C_VEL
LIN {X 0,Y 303.612,Z 582.751,A -85,B 0,C 180,E1 -17047.003,E2 -17047.003} C_VEL
LIN {X 0,Y 302.11,Z 580.887,A -85,B 0,C 180,E1 -17049.854,E2 -17049.854} C_VEL
LIN {X 0,Y 301.459,Z 580.449,A -85,B 0,C 180,E1 -17052.54,E2 -17052.54} C_VEL
LIN {X 0,Y 301.439,Z 580.842,A -85,B 0,C 180,E1 -17054.384,E2 -17054.384} C_VEL
LIN {X 0,Y 301.575,Z 581.939,A -85,B 0,C 180,E1 -17056.257,E2 -17056.257} C_VEL
LIN {X 0,Y 301.973,Z 583.617,A -85,B 0,C 180,E1 -17058.139,E2 -17058.139} C_VEL
LIN {X 0,Y 302.853,Z 587.821,A -85,B 0,C 180,E1 -17061.203,E2 -17061.203} C_VEL
LIN {X 0,Y 303.823,Z 593.278,A -85,B 0,C 180,E1 -17064.06,E2 -17064.06} C_VEL
LIN {X 0,Y 304.436,Z 598.883,A -85,B 0,C 180,E1 -17066.355,E2 -17066.355} C_VEL
LIN {X 0,Y 304.651,Z 602.179,A -85,B 0,C 180,E1 -17067.536,E2 -17067.536} C_VEL
LIN {X 0,Y 302.354,Z 611.543,A -85,B 0,C 180,E1 -17069.823,E2 -17069.823} C_VEL
LIN {X 0,Y 300.966,Z 618.135,A -85,B 0,C 180,E1 -17071.328,E2 -17071.328} C_VEL
LIN {X 0,Y 303.278,Z 630.909,A -85,B 0,C 180,E1 -17072.803,E2 -17072.803} C_VEL
LIN {X 0,Y 305.315,Z 644.901,A -85,B 0,C 180,E1 -17074.134,E2 -17074.134} C_VEL
LIN {X 0,Y 305.865,Z 651.371,A -85,B 0,C 180,E1 -17074.649,E2 -17074.649} C_VEL
LIN {X 0,Y 301.057,Z 701.615,A -85,B 0,C 180,E1 -17076.755,E2 -17076.755} C_VEL
LIN {X 0,Y 299.468,Z 713.58,A -85,B 0,C 180,E1 -17077.491,E2 -17077.491} C_VEL
LIN {X 0,Y 297.522,Z 725.199,A -85,B 0,C 180,E1 -17078.522,E2 -17078.522} C_VEL
LIN {X 0,Y 295.567,Z 735.176,A -85,B 0,C 180,E1 -17079.65,E2 -17079.65} C_VEL
LIN {X 0,Y 293.278,Z 745.224,A -85,B 0,C 180,E1 -17081.125,E2 -17081.125} C_VEL
LIN {X 0,Y 291.412,Z 752.432,A -85,B 0,C 180,E1 -17082.454,E2 -17082.454} C_VEL
LIN {X 0,Y 289.796,Z 758.43,A -85,B 0,C 180,E1 -17083.806,E2 -17083.806} C_VEL
LIN {X 0,Y 288.069,Z 764.661,A -85,B 0,C 180,E1 -17085.518,E2 -17085.518} C_VEL
LIN {X 0,Y 286.479,Z 769.681,A -85,B 0,C 180,E1 -17087.245,E2 -17087.245} C_VEL
LIN {X 0,Y 284.947,Z 774.195,A -85,B 0,C 180,E1 -17089.34,E2 -17089.34} C_VEL
LIN {X 0,Y 283.874,Z 777.304,A -85,B 0,C 180,E1 -17091.457,E2 -17091.457} C_VEL
LIN {X 0,Y 283.379,Z 778.739,A -85,B 0,C 180,E1 -17092.877,E2 -17092.877} C_VEL
LIN {X 0,Y 282.953,Z 779.654,A -85,B 0,C 180,E1 -17094.298,E2 -17094.298} C_VEL
LIN {X 0,Y 282.622,Z 779.973,A -85,B 0,C 180,E1 -17095.722,E2 -17095.722} C_VEL
LIN {X 0,Y 282.413,Z 779.722,A -85,B 0,C 180,E1 -17097.147,E2 -17097.147} C_VEL
LIN {X 0,Y 282.321,Z 778.964,A -85,B 0,C 180,E1 -17098.574,E2 -17098.574} C_VEL
LIN {X 0,Y 282.296,Z 777.686,A -85,B 0,C 180,E1 -17100,E2 -17100} C_VEL
LIN {X 0,Y 282.354,Z 774.634,A -85,B 0,C 180,E1 -17102.14,E2 -17102.14} C_VEL
LIN {X 0,Y 282.525,Z 771.831,A -85,B 0,C 180,E1 -17103.566,E2 -17103.566} C_VEL
LIN {X 0,Y 282.566,Z 767.654,A -85,B 0,C 180,E1 -17105.237,E2 -17105.237} C_VEL
LIN {X 0,Y 282.923,Z 761.662,A -85,B 0,C 180,E1 -17107.135,E2 -17107.135} C_VEL
LIN {X 0,Y 283.257,Z 754.418,A -85,B 0,C 180,E1 -17108.921,E2 -17108.921} C_VEL
LIN {X 0,Y 283.746,Z 746.244,A -85,B 0,C 180,E1 -17110.525,E2 -17110.525} C_VEL
LIN {X 0,Y 284.359,Z 737.352,A -85,B 0,C 180,E1 -17111.946,E2 -17111.946} C_VEL
LIN {X 0,Y 284.947,Z 727.494,A -85,B 0,C 180,E1 -17113.188,E2 -17113.188} C_VEL
LIN {X 0,Y 285.547,Z 716.558,A -85,B 0,C 180,E1 -17114.248,E2 -17114.248} C_VEL
LIN {X 0,Y 285.903,Z 705.628,A -85,B 0,C 180,E1 -17115.049,E2 -17115.049} C_VEL
LIN {X 0,Y 286.428,Z 692.851,A -85,B 0,C 180,E1 -17115.659,E2 -17115.659} C_VEL
LIN {X 0,Y 287.643,Z 641.451,A -85,B 0,C 180,E1 -17117.575,E2 -17117.575} C_VEL
LIN {X 0,Y 285.863,Z 619.554,A -85,B 0,C 180,E1 -17118.457,E2 -17118.457} C_VEL
LIN {X 0,Y 285.786,Z 617.077,A -85,B 0,C 180,E1 -17118.599,E2 -17118.599} C_VEL
LIN {X 0,Y 287.233,Z 597.671,A -85,B 0,C 180,E1 -17122.667,E2 -17122.667} C_VEL
LIN {X 0,Y 288.837,Z 578.228,A -85,B 0,C 180,E1 -17126.753,E2 -17126.753} C_VEL
LIN {X 0,Y 289.167,Z 572.994,A -85,B 0,C 180,E1 -17127.86,E2 -17127.86} C_VEL
LIN {X 0,Y 287.255,Z 563.075,A -85,B 0,C 180,E1 -17130.103,E2 -17130.103} C_VEL
LIN {X 0,Y 284.409,Z 549.194,A -85,B 0,C 180,E1 -17133.354,E2 -17133.354} C_VEL
LIN {X 0,Y 284.355,Z 549.065,A -85,B 0,C 180,E1 -17136.383,E2 -17136.383} C_VEL
LIN {X 0,Y 284.31,Z 549.04,A -85,B 0,C 180,E1 -17139.994,E2 -17139.994} C_VEL
LIN {X 0,Y 284.249,Z 549.041,A -85,B 0,C 180,E1 -17144.19,E2 -17144.19} C_VEL
LIN {X 0,Y 284.276,Z 549.06,A -85,B 0,C 180,E1 -17148.124,E2 -17148.124} C_VEL
LIN {X 0,Y 284.323,Z 549.051,A -85,B 0,C 180,E1 -17152.278,E2 -17152.278} C_VEL
LIN {X 0,Y 284.312,Z 549.057,A -85,B 0,C 180,E1 -17155.35,E2 -17155.35} C_VEL
LIN {X 0,Y 284.348,Z 549.188,A -85,B 0,C 180,E1 -17159.207,E2 -17159.207} C_VEL
LIN {X 0,Y 285.615,Z 554.593,A -85,B 0,C 180,E1 -17161.345,E2 -17161.345} C_VEL
LIN {X 0,Y 288.548,Z 561.058,A -85,B 0,C 180,E1 -17161.904,E2 -17161.904} C_VEL
LIN {X 0,Y 296.09,Z 579.024,A -85,B 0,C 180,E1 -17163.168,E2 -17163.168} C_VEL
LIN {X 0,Y 298.162,Z 585.126,A -85,B 0,C 180,E1 -17163.533,E2 -17163.533} C_VEL
LIN {X 0,Y 298.975,Z 589.528,A -85,B 0,C 180,E1 -17163.727,E2 -17163.727} C_VEL
LIN {X 0,Y 296.964,Z 659.438,A -85,B 0,C 180,E1 -17165.393,E2 -17165.393} C_VEL
LIN {X 0,Y 296.383,Z 671.941,A -85,B 0,C 180,E1 -17165.901,E2 -17165.901} C_VEL
LIN {X 0,Y 295.238,Z 684.734,A -85,B 0,C 180,E1 -17166.686,E2 -17166.686} C_VEL
LIN {X 0,Y 293.898,Z 696.566,A -85,B 0,C 180,E1 -17167.689,E2 -17167.689} C_VEL
LIN {X 0,Y 292.39,Z 707.312,A -85,B 0,C 180,E1 -17168.865,E2 -17168.865} C_VEL
LIN {X 0,Y 290.849,Z 717.193,A -85,B 0,C 180,E1 -17170.226,E2 -17170.226} C_VEL
LIN {X 0,Y 289.264,Z 727.154,A -85,B 0,C 180,E1 -17171.953,E2 -17171.953} C_VEL
LIN {X 0,Y 287.399,Z 736.795,A -85,B 0,C 180,E1 -17174.031,E2 -17174.031} C_VEL
LIN {X 0,Y 285.911,Z 744.477,A -85,B 0,C 180,E1 -17176.132,E2 -17176.132} C_VEL
LIN {X 0,Y 284.519,Z 751.531,A -85,B 0,C 180,E1 -17178.602,E2 -17178.602} C_VEL
LIN {X 0,Y 283.609,Z 756.228,A -85,B 0,C 180,E1 -17180.73,E2 -17180.73} C_VEL
LIN {X 0,Y 283.054,Z 759.814,A -85,B 0,C 180,E1 -17182.867,E2 -17182.867} C_VEL
LIN {X 0,Y 282.799,Z 761.667,A -85,B 0,C 180,E1 -17184.294,E2 -17184.294} C_VEL
LIN {X 0,Y 282.63,Z 763.061,A -85,B 0,C 180,E1 -17185.721,E2 -17185.721} C_VEL
LIN {X 0,Y 282.493,Z 764.055,A -85,B 0,C 180,E1 -17187.147,E2 -17187.147} C_VEL
LIN {X 0,Y 282.364,Z 764.898,A -85,B 0,C 180,E1 -17189.999,E2 -17189.999} C_VEL
LIN {X 0,Y 282.38,Z 764.707,A -85,B 0,C 180,E1 -17191.425,E2 -17191.425} C_VEL
LIN {X 0,Y 282.491,Z 764.121,A -85,B 0,C 180,E1 -17192.851,E2 -17192.851} C_VEL
LIN {X 0,Y 282.625,Z 763.156,A -85,B 0,C 180,E1 -17194.277,E2 -17194.277} C_VEL
LIN {X 0,Y 282.946,Z 760.817,A -85,B 0,C 180,E1 -17196.509,E2 -17196.509} C_VEL
LIN {X 0,Y 283.396,Z 757.737,A -85,B 0,C 180,E1 -17198.556,E2 -17198.556} C_VEL
LIN {X 0,Y 284.131,Z 753.485,A -85,B 0,C 180,E1 -17200.69,E2 -17200.69} C_VEL
LIN {X 0,Y 285.397,Z 747.048,A -85,B 0,C 180,E1 -17203.165,E2 -17203.165} C_VEL
LIN {X 0,Y 286.722,Z 739.97,A -85,B 0,C 180,E1 -17205.276,E2 -17205.276} C_VEL
LIN {X 0,Y 288.594,Z 731.144,A -85,B 0,C 180,E1 -17207.355,E2 -17207.355} C_VEL
LIN {X 0,Y 290.236,Z 721.447,A -85,B 0,C 180,E1 -17209.199,E2 -17209.199} C_VEL
LIN {X 0,Y 291.862,Z 710.778,A -85,B 0,C 180,E1 -17210.803,E2 -17210.803} C_VEL
LIN {X 0,Y 293.565,Z 699.328,A -85,B 0,C 180,E1 -17212.15,E2 -17212.15} C_VEL
LIN {X 0,Y 295.06,Z 687.303,A -85,B 0,C 180,E1 -17213.233,E2 -17213.233} C_VEL
LIN {X 0,Y 296.156,Z 674.661,A -85,B 0,C 180,E1 -17214.07,E2 -17214.07} C_VEL
LIN {X 0,Y 296.927,Z 661.522,A -85,B 0,C 180,E1 -17214.654,E2 -17214.654} C_VEL
LIN {X 0,Y 298.611,Z 605.382,A -85,B 0,C 180,E1 -17216.009,E2 -17216.009} C_VEL
LIN {X 0,Y 298.861,Z 588.456,A -85,B 0,C 180,E1 -17216.43,E2 -17216.43} C_VEL
LIN {X 0,Y 297.491,Z 582.731,A -85,B 0,C 180,E1 -17216.714,E2 -17216.714} C_VEL
LIN {X 0,Y 289.977,Z 564.164,A -85,B 0,C 180,E1 -17217.979,E2 -17217.979} C_VEL
LIN {X 0,Y 285.638,Z 554.659,A -85,B 0,C 180,E1 -17218.766,E2 -17218.766} C_VEL
LIN {X 0,Y 284.337,Z 549.259,A -85,B 0,C 180,E1 -17220.878,E2 -17220.878} C_VEL
LIN {X 0,Y 284.342,Z 549.062,A -85,B 0,C 180,E1 -17225.113,E2 -17225.113} C_VEL
LIN {X 0,Y 284.324,Z 549.068,A -85,B 0,C 180,E1 -17228.165,E2 -17228.165} C_VEL
LIN {X 0,Y 284.246,Z 549.071,A -85,B 0,C 180,E1 -17231.226,E2 -17231.226} C_VEL
LIN {X 0,Y 283.601,Z 549.162,A -85,B 0,C 180,E1 -17232.409,E2 -17232.409} C_VEL
LIN {X 0,Y 280.784,Z 549.519,A -85,B 0,C 180,E1 -17234.337,E2 -17234.337} C_VEL
LIN {X 0,Y 278.372,Z 549.815,A -85,B 0,C 180,E1 -17235.902,E2 -17235.902} C_VEL
LIN {X 0,Y 277.318,Z 549.94,A -85,B 0,C 180,E1 -17237.115,E2 -17237.115} C_VEL
LIN {X 0,Y 277.222,Z 549.95,A -85,B 0,C 180,E1 -17237.526,E2 -17237.526} C_VEL
LIN {X 0,Y 277.261,Z 549.922,A -85,B 0,C 180,E1 -17240.676,E2 -17240.676} C_VEL
LIN {X 0,Y 277.315,Z 549.94,A -85,B 0,C 180,E1 -17244.346,E2 -17244.346} C_VEL
LIN {X 0,Y 277.239,Z 549.944,A -85,B 0,C 180,E1 -17247.835,E2 -17247.835} C_VEL
LIN {X 0,Y 277.284,Z 549.94,A -85,B 0,C 180,E1 -17251.212,E2 -17251.212} C_VEL
LIN {X 0,Y 277.308,Z 549.941,A -85,B 0,C 180,E1 -17254.479,E2 -17254.479} C_VEL
LIN {X 0,Y 277.279,Z 549.933,A -85,B 0,C 180,E1 -17257.654,E2 -17257.654} C_VEL
LIN {X 0,Y 277.339,Z 549.936,A -85,B 0,C 180,E1 -17260.766,E2 -17260.766} C_VEL
LIN {X 0,Y 277.428,Z 549.919,A -85,B 0,C 180,E1 -17265.325,E2 -17265.325} C_VEL
LIN {X 0,Y 277.5,Z 549.902,A -85,B 0,C 180,E1 -17269.788,E2 -17269.788} C_VEL
LIN {X 0,Y 277.646,Z 549.897,A -85,B 0,C 180,E1 -17272.729,E2 -17272.729} C_VEL
LIN {X 0,Y 277.816,Z 549.873,A -85,B 0,C 180,E1 -17278.55,E2 -17278.55} C_VEL
LIN {X 0,Y 277.816,Z 549.876,A -85,B 0,C 180,E1 -17281.45,E2 -17281.45} C_VEL
LIN {X 0,Y 277.647,Z 549.901,A -85,B 0,C 180,E1 -17287.271,E2 -17287.271} C_VEL
LIN {X 0,Y 277.5,Z 549.902,A -85,B 0,C 180,E1 -17290.212,E2 -17290.212} C_VEL
LIN {X 0,Y 277.428,Z 549.922,A -85,B 0,C 180,E1 -17294.674,E2 -17294.674} C_VEL
LIN {X 0,Y 277.34,Z 549.939,A -85,B 0,C 180,E1 -17299.234,E2 -17299.234} C_VEL
LIN {X 0,Y 277.312,Z 549.942,A -85,B 0,C 180,E1 -17304.171,E2 -17304.171} C_VEL
LIN {X 0,Y 277.314,Z 549.934,A -85,B 0,C 180,E1 -17307.504,E2 -17307.504} C_VEL
LIN {X 0,Y 277.266,Z 549.942,A -85,B 0,C 180,E1 -17310.482,E2 -17310.482} C_VEL
LIN {X 0,Y 277.241,Z 549.947,A -85,B 0,C 180,E1 -17313.897,E2 -17313.897} C_VEL
LIN {X 0,Y 277.262,Z 549.925,A -85,B 0,C 180,E1 -17317.47,E2 -17317.47} C_VEL
LIN {X 0,Y 277.228,Z 549.942,A -85,B 0,C 180,E1 -17321.233,E2 -17321.233} C_VEL
LIN {X 0,Y 277.242,Z 549.952,A -85,B 0,C 180,E1 -17325.218,E2 -17325.218} C_VEL
LIN {X 0,Y 277.291,Z 549.942,A -85,B 0,C 180,E1 -17329.496,E2 -17329.496} C_VEL
LIN {X 0,Y 277.315,Z 549.989,A -85,B 0,C 180,E1 -17333.937,E2 -17333.937} C_VEL
LIN {X 0,Y 279.575,Z 559.685,A -85,B 0,C 180,E1 -17337.713,E2 -17337.713} C_VEL
LIN {X 0,Y 281.436,Z 568.37,A -85,B 0,C 180,E1 -17340.783,E2 -17340.783} C_VEL
LIN {X 0,Y 284.131,Z 574.995,A -85,B 0,C 180,E1 -17341.333,E2 -17341.333} C_VEL
LIN {X 0,Y 286.954,Z 582.558,A -85,B 0,C 180,E1 -17341.849,E2 -17341.849} C_VEL
LIN {X 0,Y 291.511,Z 610.368,A -85,B 0,C 180,E1 -17343.077,E2 -17343.077} C_VEL
LIN {X 0,Y 292.078,Z 615.328,A -85,B 0,C 180,E1 -17343.267,E2 -17343.267} C_VEL
LIN {X 0,Y 290.242,Z 676.926,A -85,B 0,C 180,E1 -17344.786,E2 -17344.786} C_VEL
LIN {X 0,Y 289.12,Z 690.834,A -85,B 0,C 180,E1 -17345.402,E2 -17345.402} C_VEL
LIN {X 0,Y 287.807,Z 703.287,A -85,B 0,C 180,E1 -17346.241,E2 -17346.241} C_VEL
LIN {X 0,Y 286.325,Z 714.402,A -85,B 0,C 180,E1 -17347.259,E2 -17347.259} C_VEL
LIN {X 0,Y 284.47,Z 725.973,A -85,B 0,C 180,E1 -17348.63,E2 -17348.63} C_VEL
LIN {X 0,Y 282.62,Z 736.394,A -85,B 0,C 180,E1 -17350.197,E2 -17350.197} C_VEL
LIN {X 0,Y 280.958,Z 745.503,A -85,B 0,C 180,E1 -17351.907,E2 -17351.907} C_VEL
LIN {X 0,Y 279.276,Z 754.164,A -85,B 0,C 180,E1 -17353.931,E2 -17353.931} C_VEL
LIN {X 0,Y 277.824,Z 761.597,A -85,B 0,C 180,E1 -17356.096,E2 -17356.096} C_VEL
LIN {X 0,Y 276.714,Z 767.566,A -85,B 0,C 180,E1 -17358.278,E2 -17358.278} C_VEL
LIN {X 0,Y 275.962,Z 772.287,A -85,B 0,C 180,E1 -17360.473,E2 -17360.473} C_VEL
LIN {X 0,Y 275.495,Z 775.9,A -85,B 0,C 180,E1 -17362.673,E2 -17362.673} C_VEL
LIN {X 0,Y 275.263,Z 778.341,A -85,B 0,C 180,E1 -17364.715,E2 -17364.715} C_VEL
LIN {X 0,Y 275.255,Z 780.158,A -85,B 0,C 180,E1 -17367.074,E2 -17367.074} C_VEL
LIN {X 0,Y 275.239,Z 781.326,A -85,B 0,C 180,E1 -17370.001,E2 -17370.001} C_VEL
LIN {X 0,Y 275.241,Z 782.724,A -85,B 0,C 180,E1 -17371.464,E2 -17371.464} C_VEL
LIN {X 0,Y 275.27,Z 783.631,A -85,B 0,C 180,E1 -17372.928,E2 -17372.928} C_VEL
LIN {X 0,Y 275.317,Z 783.939,A -85,B 0,C 180,E1 -17374.393,E2 -17374.393} C_VEL
LIN {X 0,Y 275.495,Z 783.664,A -85,B 0,C 180,E1 -17375.858,E2 -17375.858} C_VEL
LIN {X 0,Y 275.713,Z 782.891,A -85,B 0,C 180,E1 -17377.324,E2 -17377.324} C_VEL
LIN {X 0,Y 276.151,Z 781.61,A -85,B 0,C 180,E1 -17378.785,E2 -17378.785} C_VEL
LIN {X 0,Y 277.1,Z 778.606,A -85,B 0,C 180,E1 -17380.967,E2 -17380.967} C_VEL
LIN {X 0,Y 277.859,Z 775.917,A -85,B 0,C 180,E1 -17382.416,E2 -17382.416} C_VEL
LIN {X 0,Y 279.262,Z 770.667,A -85,B 0,C 180,E1 -17384.577,E2 -17384.577} C_VEL
LIN {X 0,Y 281.235,Z 763.77,A -85,B 0,C 180,E1 -17386.702,E2 -17386.702} C_VEL
LIN {X 0,Y 282.969,Z 756.492,A -85,B 0,C 180,E1 -17388.463,E2 -17388.463} C_VEL
LIN {X 0,Y 284.703,Z 748.479,A -85,B 0,C 180,E1 -17390.031,E2 -17390.031} C_VEL
LIN {X 0,Y 286.642,Z 738.641,A -85,B 0,C 180,E1 -17391.58,E2 -17391.58} C_VEL
LIN {X 0,Y 288.238,Z 729.021,A -85,B 0,C 180,E1 -17392.774,E2 -17392.774} C_VEL
LIN {X 0,Y 289.705,Z 718.71,A -85,B 0,C 180,E1 -17393.786,E2 -17393.786} C_VEL
LIN {X 0,Y 291.034,Z 706.041,A -85,B 0,C 180,E1 -17394.714,E2 -17394.714} C_VEL
LIN {X 0,Y 292.653,Z 686.068,A -85,B 0,C 180,E1 -17395.756,E2 -17395.756} C_VEL
LIN {X 0,Y 300.299,Z 618.027,A -85,B 0,C 180,E1 -17398.824,E2 -17398.824} C_VEL
LIN {X 0,Y 300.793,Z 614.252,A -85,B 0,C 180,E1 -17399.253,E2 -17399.253} C_VEL
LIN {X 0,Y 302.596,Z 605.566,A -85,B 0,C 180,E1 -17400.43,E2 -17400.43} C_VEL
LIN {X 0,Y 302.883,Z 602.289,A -85,B 0,C 180,E1 -17401.051,E2 -17401.051} C_VEL
LIN {X 0,Y 302.399,Z 596.482,A -85,B 0,C 180,E1 -17402.65,E2 -17402.65} C_VEL
LIN {X 0,Y 302.114,Z 593.739,A -85,B 0,C 180,E1 -17403.554,E2 -17403.554} C_VEL
LIN {X 0,Y 300.84,Z 590.833,A -85,B 0,C 180,E1 -17405.15,E2 -17405.15} C_VEL
LIN {X 0,Y 299.052,Z 587.943,A -85,B 0,C 180,E1 -17407.665,E2 -17407.665} C_VEL
LIN {X 0,Y 298.027,Z 586.75,A -85,B 0,C 180,E1 -17409.548,E2 -17409.548} C_VEL
LIN {X 0,Y 297.368,Z 586.191,A -85,B 0,C 180,E1 -17411.435,E2 -17411.435} C_VEL
LIN {X 0,Y 297.071,Z 586.178,A -85,B 0,C 180,E1 -17413.321,E2 -17413.321} C_VEL
LIN {X 0,Y 297.041,Z 586.826,A -85,B 0,C 180,E1 -17415.22,E2 -17415.22} C_VEL
LIN {X 0,Y 297.179,Z 588.173,A -85,B 0,C 180,E1 -17417.15,E2 -17417.15} C_VEL
LIN {X 0,Y 297.525,Z 590.233,A -85,B 0,C 180,E1 -17419.104,E2 -17419.104} C_VEL
LIN {X 0,Y 298.003,Z 593.028,A -85,B 0,C 180,E1 -17421.103,E2 -17421.103} C_VEL
LIN {X 0,Y 298.743,Z 598.385,A -85,B 0,C 180,E1 -17423.975,E2 -17423.975} C_VEL
LIN {X 0,Y 299.176,Z 604.027,A -85,B 0,C 180,E1 -17426.332,E2 -17426.332} C_VEL
LIN {X 0,Y 299.036,Z 606.824,A -85,B 0,C 180,E1 -17427.279,E2 -17427.279} C_VEL
LIN {X 0,Y 296.086,Z 617.942,A -85,B 0,C 180,E1 -17429.979,E2 -17429.979} C_VEL
LIN {X 0,Y 298.482,Z 631.961,A -85,B 0,C 180,E1 -17431.722,E2 -17431.722} C_VEL
LIN {X 0,Y 300.422,Z 646.951,A -85,B 0,C 180,E1 -17433.246,E2 -17433.246} C_VEL
LIN {X 0,Y 300.894,Z 652.427,A -85,B 0,C 180,E1 -17433.702,E2 -17433.702} C_VEL
LIN {X 0,Y 295.77,Z 701.806,A -85,B 0,C 180,E1 -17435.849,E2 -17435.849} C_VEL
LIN {X 0,Y 294.112,Z 713.729,A -85,B 0,C 180,E1 -17436.593,E2 -17436.593} C_VEL
LIN {X 0,Y 292.182,Z 724.578,A -85,B 0,C 180,E1 -17437.552,E2 -17437.552} C_VEL
LIN {X 0,Y 290.38,Z 733.218,A -85,B 0,C 180,E1 -17438.527,E2 -17438.527} C_VEL
LIN {X 0,Y 288.384,Z 741.539,A -85,B 0,C 180,E1 -17439.679,E2 -17439.679} C_VEL
LIN {X 0,Y 285.8,Z 751.164,A -85,B 0,C 180,E1 -17441.357,E2 -17441.357} C_VEL
LIN {X 0,Y 284.006,Z 757.395,A -85,B 0,C 180,E1 -17442.725,E2 -17442.725} C_VEL
LIN {X 0,Y 282.376,Z 762.63,A -85,B 0,C 180,E1 -17444.111,E2 -17444.111} C_VEL
LIN {X 0,Y 280.987,Z 767.013,A -85,B 0,C 180,E1 -17445.516,E2 -17445.516} C_VEL
LIN {X 0,Y 279.058,Z 772.224,A -85,B 0,C 180,E1 -17447.639,E2 -17447.639} C_VEL
LIN {X 0,Y 278.031,Z 774.914,A -85,B 0,C 180,E1 -17449.072,E2 -17449.072} C_VEL
LIN {X 0,Y 276.88,Z 777.837,A -85,B 0,C 180,E1 -17451.24,E2 -17451.24} C_VEL
LIN {X 0,Y 276.339,Z 779.075,A -85,B 0,C 180,E1 -17452.694,E2 -17452.694} C_VEL
LIN {X 0,Y 275.892,Z 779.814,A -85,B 0,C 180,E1 -17454.152,E2 -17454.152} C_VEL
LIN {X 0,Y 275.539,Z 780.051,A -85,B 0,C 180,E1 -17455.612,E2 -17455.612} C_VEL
LIN {X 0,Y 275.331,Z 779.693,A -85,B 0,C 180,E1 -17457.074,E2 -17457.074} C_VEL
LIN {X 0,Y 275.249,Z 778.76,A -85,B 0,C 180,E1 -17458.537,E2 -17458.537} C_VEL
LIN {X 0,Y 275.209,Z 776.436,A -85,B 0,C 180,E1 -17460.732,E2 -17460.732} C_VEL
LIN {X 0,Y 275.377,Z 772.688,A -85,B 0,C 180,E1 -17462.926,E2 -17462.926} C_VEL
LIN {X 0,Y 275.479,Z 768.297,A -85,B 0,C 180,E1 -17464.805,E2 -17464.805} C_VEL
LIN {X 0,Y 275.719,Z 763.208,A -85,B 0,C 180,E1 -17466.513,E2 -17466.513} C_VEL
LIN {X 0,Y 276.018,Z 757.585,A -85,B 0,C 180,E1 -17468.05,E2 -17468.05} C_VEL
LIN {X 0,Y 276.47,Z 749.351,A -85,B 0,C 180,E1 -17469.88,E2 -17469.88} C_VEL
LIN {X 0,Y 276.985,Z 740.995,A -85,B 0,C 180,E1 -17471.341,E2 -17471.341} C_VEL
LIN {X 0,Y 277.561,Z 732.053,A -85,B 0,C 180,E1 -17472.615,E2 -17472.615} C_VEL
LIN {X 0,Y 278.253,Z 720.794,A -85,B 0,C 180,E1 -17473.884,E2 -17473.884} C_VEL
LIN {X 0,Y 278.766,Z 709.808,A -85,B 0,C 180,E1 -17474.789,E2 -17474.789} C_VEL
LIN {X 0,Y 279.052,Z 698.431,A -85,B 0,C 180,E1 -17475.474,E2 -17475.474} C_VEL
LIN {X 0,Y 280.252,Z 658.86,A -85,B 0,C 180,E1 -17477.043,E2 -17477.043} C_VEL
LIN {X 0,Y 280.489,Z 641.055,A -85,B 0,C 180,E1 -17477.745,E2 -17477.745} C_VEL
LIN {X 0,Y 278.756,Z 618.601,A -85,B 0,C 180,E1 -17478.66,E2 -17478.66} C_VEL
LIN {X 0,Y 278.781,Z 616.865,A -85,B 0,C 180,E1 -17478.816,E2 -17478.816} C_VEL
LIN {X 0,Y 280.338,Z 596.1,A -85,B 0,C 180,E1 -17483.257,E2 -17483.257} C_VEL
LIN {X 0,Y 282.023,Z 576.484,A -85,B 0,C 180,E1 -17487.453,E2 -17487.453} C_VEL
LIN {X 0,Y 282.033,Z 572.788,A -85,B 0,C 180,E1 -17488.259,E2 -17488.259} C_VEL
LIN {X 0,Y 278.334,Z 554.932,A -85,B 0,C 180,E1 -17492.409,E2 -17492.409} C_VEL
LIN {X 0,Y 277.367,Z 550.075,A -85,B 0,C 180,E1 -17493.603,E2 -17493.603} C_VEL
LIN {X 0,Y 277.286,Z 549.947,A -85,B 0,C 180,E1 -17497.467,E2 -17497.467} C_VEL
LIN {X 0,Y 277.213,Z 549.901,A -85,B 0,C 180,E1 -17501.236,E2 -17501.236} C_VEL
LIN {X 0,Y 277.205,Z 549.942,A -85,B 0,C 180,E1 -17505.226,E2 -17505.226} C_VEL
LIN {X 0,Y 277.226,Z 549.916,A -85,B 0,C 180,E1 -17509.512,E2 -17509.512} C_VEL
LIN {X 0,Y 277.269,Z 549.934,A -85,B 0,C 180,E1 -17512.53,E2 -17512.53} C_VEL
LIN {X 0,Y 277.251,Z 549.938,A -85,B 0,C 180,E1 -17516.104,E2 -17516.104} C_VEL
LIN {X 0,Y 277.297,Z 550.059,A -85,B 0,C 180,E1 -17518.59,E2 -17518.59} C_VEL
LIN {X 0,Y 278.456,Z 554.867,A -85,B 0,C 180,E1 -17520.545,E2 -17520.545} C_VEL
LIN {X 0,Y 282.63,Z 563.932,A -85,B 0,C 180,E1 -17521.338,E2 -17521.338} C_VEL
LIN {X 0,Y 289.559,Z 580.381,A -85,B 0,C 180,E1 -17522.544,E2 -17522.544} C_VEL
LIN {X 0,Y 292.051,Z 587.524,A -85,B 0,C 180,E1 -17522.993,E2 -17522.993} C_VEL
LIN {X 0,Y 292.601,Z 590.731,A -85,B 0,C 180,E1 -17523.136,E2 -17523.136} C_VEL
LIN {X 0,Y 290.526,Z 659.663,A -85,B 0,C 180,E1 -17524.81,E2 -17524.81} C_VEL
LIN {X 0,Y 289.912,Z 672.157,A -85,B 0,C 180,E1 -17525.327,E2 -17525.327} C_VEL
LIN {X 0,Y 288.734,Z 684.946,A -85,B 0,C 180,E1 -17526.129,E2 -17526.129} C_VEL
LIN {X 0,Y 287.367,Z 696.776,A -85,B 0,C 180,E1 -17527.153,E2 -17527.153} C_VEL
LIN {X 0,Y 285.791,Z 707.521,A -85,B 0,C 180,E1 -17528.353,E2 -17528.353} C_VEL
LIN {X 0,Y 284.185,Z 717.401,A -85,B 0,C 180,E1 -17529.742,E2 -17529.742} C_VEL
LIN {X 0,Y 282.523,Z 727.362,A -85,B 0,C 180,E1 -17531.507,E2 -17531.507} C_VEL
LIN {X 0,Y 280.595,Z 737.002,A -85,B 0,C 180,E1 -17533.633,E2 -17533.633} C_VEL
LIN {X 0,Y 278.991,Z 744.685,A -85,B 0,C 180,E1 -17535.781,E2 -17535.781} C_VEL
LIN {X 0,Y 277.542,Z 751.738,A -85,B 0,C 180,E1 -17538.311,E2 -17538.311} C_VEL
LIN {X 0,Y 276.585,Z 756.434,A -85,B 0,C 180,E1 -17540.492,E2 -17540.492} C_VEL
LIN {X 0,Y 276.009,Z 760.02,A -85,B 0,C 180,E1 -17542.684,E2 -17542.684} C_VEL
LIN {X 0,Y 275.724,Z 761.873,A -85,B 0,C 180,E1 -17544.147,E2 -17544.147} C_VEL
LIN {X 0,Y 275.557,Z 763.266,A -85,B 0,C 180,E1 -17545.611,E2 -17545.611} C_VEL
LIN {X 0,Y 275.427,Z 764.259,A -85,B 0,C 180,E1 -17547.073,E2 -17547.073} C_VEL
LIN {X 0,Y 275.286,Z 765.102,A -85,B 0,C 180,E1 -17549.999,E2 -17549.999} C_VEL
LIN {X 0,Y 275.306,Z 764.911,A -85,B 0,C 180,E1 -17551.462,E2 -17551.462} C_VEL
LIN {X 0,Y 275.424,Z 764.325,A -85,B 0,C 180,E1 -17552.924,E2 -17552.924} C_VEL
LIN {X 0,Y 275.552,Z 763.36,A -85,B 0,C 180,E1 -17554.387,E2 -17554.387} C_VEL
LIN {X 0,Y 275.861,Z 761.246,A -85,B 0,C 180,E1 -17556.49,E2 -17556.49} C_VEL
LIN {X 0,Y 276.386,Z 757.941,A -85,B 0,C 180,E1 -17558.775,E2 -17558.775} C_VEL
LIN {X 0,Y 277.15,Z 753.689,A -85,B 0,C 180,E1 -17560.962,E2 -17560.962} C_VEL
LIN {X 0,Y 278.495,Z 747.25,A -85,B 0,C 180,E1 -17563.498,E2 -17563.498} C_VEL
LIN {X 0,Y 279.884,Z 740.172,A -85,B 0,C 180,E1 -17565.659,E2 -17565.659} C_VEL
LIN {X 0,Y 281.84,Z 731.346,A -85,B 0,C 180,E1 -17567.785,E2 -17567.785} C_VEL
LIN {X 0,Y 283.546,Z 721.622,A -85,B 0,C 180,E1 -17569.675,E2 -17569.675} C_VEL
LIN {X 0,Y 285.254,Z 710.978,A -85,B 0,C 180,E1 -17571.308,E2 -17571.308} C_VEL
LIN {X 0,Y 287.019,Z 699.527,A -85,B 0,C 180,E1 -17572.683,E2 -17572.683} C_VEL
LIN {X 0,Y 288.555,Z 687.5,A -85,B 0,C 180,E1 -17573.789,E2 -17573.789} C_VEL
LIN {X 0,Y 289.691,Z 674.856,A -85,B 0,C 180,E1 -17574.642,E2 -17574.642} C_VEL
LIN {X 0,Y 290.508,Z 661.711,A -85,B 0,C 180,E1 -17575.237,E2 -17575.237} C_VEL
LIN {X 0,Y 292.259,Z 604.223,A -85,B 0,C 180,E1 -17576.654,E2 -17576.654} C_VEL
LIN {X 0,Y 292.558,Z 589.849,A -85,B 0,C 180,E1 -17577.012,E2 -17577.012} C_VEL
LIN {X 0,Y 291.498,Z 585.385,A -85,B 0,C 180,E1 -17577.241,E2 -17577.241} C_VEL
LIN {X 0,Y 284.212,Z 567.439,A -85,B 0,C 180,E1 -17578.51,E2 -17578.51} C_VEL
LIN {X 0,Y 278.491,Z 554.972,A -85,B 0,C 180,E1 -17579.565,E2 -17579.565} C_VEL
LIN {X 0,Y 277.736,Z 552.086,A -85,B 0,C 180,E1 -17580.643,E2 -17580.643} C_VEL
LIN {X 0,Y 277.276,Z 549.963,A -85,B 0,C 180,E1 -17581.676,E2 -17581.676} C_VEL
LIN {X 0,Y 277.323,Z 549.932,A -85,B 0,C 180,E1 -17585.81,E2 -17585.81} C_VEL
LIN {X 0,Y 277.236,Z 549.939,A -85,B 0,C 180,E1 -17589.326,E2 -17589.326} C_VEL
LIN {X 0,Y 277.205,Z 549.949,A -85,B 0,C 180,E1 -17593.197,E2 -17593.197} C_VEL
LIN {X 0,Y 277.222,Z 549.95,A -85,B 0,C 180,E1 -17597.526,E2 -17597.526} C_VEL
LIN {X 0,Y 276.545,Z 550.036,A -85,B 0,C 180,E1 -17598.738,E2 -17598.738} C_VEL
LIN {X 0,Y 273.753,Z 550.373,A -85,B 0,C 180,E1 -17600.717,E2 -17600.717} C_VEL
LIN {X 0,Y 271.379,Z 550.669,A -85,B 0,C 180,E1 -17602.323,E2 -17602.323} C_VEL
LIN {X 0,Y 270.334,Z 550.801,A -85,B 0,C 180,E1 -17603.567,E2 -17603.567} C_VEL
LIN {X 0,Y 270.233,Z 550.815,A -85,B 0,C 180,E1 -17603.988,E2 -17603.988} C_VEL
LIN {X 0,Y 270.199,Z 550.823,A -85,B 0,C 180,E1 -17606.892,E2 -17606.892} C_VEL
LIN {X 0,Y 270.223,Z 550.824,A -85,B 0,C 180,E1 -17610.386,E2 -17610.386} C_VEL
LIN {X 0,Y 270.258,Z 550.816,A -85,B 0,C 180,E1 -17613.763,E2 -17613.763} C_VEL
LIN {X 0,Y 270.227,Z 550.814,A -85,B 0,C 180,E1 -17617.038,E2 -17617.038} C_VEL
LIN {X 0,Y 270.295,Z 550.814,A -85,B 0,C 180,E1 -17620.244,E2 -17620.244} C_VEL
LIN {X 0,Y 270.396,Z 550.792,A -85,B 0,C 180,E1 -17624.935,E2 -17624.935} C_VEL
LIN {X 0,Y 270.435,Z 550.783,A -85,B 0,C 180,E1 -17629.519,E2 -17629.519} C_VEL
LIN {X 0,Y 270.604,Z 550.775,A -85,B 0,C 180,E1 -17632.539,E2 -17632.539} C_VEL
LIN {X 0,Y 270.781,Z 550.749,A -85,B 0,C 180,E1 -17638.513,E2 -17638.513} C_VEL
LIN {X 0,Y 270.781,Z 550.752,A -85,B 0,C 180,E1 -17641.487,E2 -17641.487} C_VEL
LIN {X 0,Y 270.605,Z 550.778,A -85,B 0,C 180,E1 -17647.461,E2 -17647.461} C_VEL
LIN {X 0,Y 270.435,Z 550.783,A -85,B 0,C 180,E1 -17650.481,E2 -17650.481} C_VEL
LIN {X 0,Y 270.396,Z 550.795,A -85,B 0,C 180,E1 -17655.065,E2 -17655.065} C_VEL
LIN {X 0,Y 270.296,Z 550.814,A -85,B 0,C 180,E1 -17659.756,E2 -17659.756} C_VEL
LIN {X 0,Y 270.267,Z 550.819,A -85,B 0,C 180,E1 -17664.586,E2 -17664.586} C_VEL
LIN {X 0,Y 270.263,Z 550.817,A -85,B 0,C 180,E1 -17667.91,E2 -17667.91} C_VEL
LIN {X 0,Y 270.178,Z 550.823,A -85,B 0,C 180,E1 -17671.349,E2 -17671.349} C_VEL
LIN {X 0,Y 270.196,Z 550.814,A -85,B 0,C 180,E1 -17674.906,E2 -17674.906} C_VEL
LIN {X 0,Y 270.217,Z 550.821,A -85,B 0,C 180,E1 -17678.718,E2 -17678.718} C_VEL
LIN {X 0,Y 270.19,Z 550.81,A -85,B 0,C 180,E1 -17682.555,E2 -17682.555} C_VEL
LIN {X 0,Y 270.209,Z 550.814,A -85,B 0,C 180,E1 -17686.741,E2 -17686.741} C_VEL
LIN {X 0,Y 270.245,Z 550.82,A -85,B 0,C 180,E1 -17689.449,E2 -17689.449} C_VEL
LIN {X 0,Y 270.252,Z 550.877,A -85,B 0,C 180,E1 -17693.266,E2 -17693.266} C_VEL
LIN {X 0,Y 272.164,Z 558.933,A -85,B 0,C 180,E1 -17696.537,E2 -17696.537} C_VEL
LIN {X 0,Y 274.21,Z 568.208,A -85,B 0,C 180,E1 -17699.945,E2 -17699.945} C_VEL
LIN {X 0,Y 278.37,Z 578.131,A -85,B 0,C 180,E1 -17700.778,E2 -17700.778} C_VEL
LIN {X 0,Y 280.93,Z 584.877,A -85,B 0,C 180,E1 -17701.26,E2 -17701.26} C_VEL
LIN {X 0,Y 285.405,Z 612.981,A -85,B 0,C 180,E1 -17702.531,E2 -17702.531} C_VEL
LIN {X 0,Y 285.689,Z 616.74,A -85,B 0,C 180,E1 -17702.664,E2 -17702.664} C_VEL
LIN {X 0,Y 283.844,Z 676.735,A -85,B 0,C 180,E1 -17704.177,E2 -17704.177} C_VEL
LIN {X 0,Y 282.681,Z 690.638,A -85,B 0,C 180,E1 -17704.803,E2 -17704.803} C_VEL
LIN {X 0,Y 281.329,Z 703.089,A -85,B 0,C 180,E1 -17705.659,E2 -17705.659} C_VEL
LIN {X 0,Y 279.78,Z 714.202,A -85,B 0,C 180,E1 -17706.696,E2 -17706.696} C_VEL
LIN {X 0,Y 277.866,Z 725.772,A -85,B 0,C 180,E1 -17708.097,E2 -17708.097} C_VEL
LIN {X 0,Y 275.923,Z 736.192,A -85,B 0,C 180,E1 -17709.695,E2 -17709.695} C_VEL
LIN {X 0,Y 274.062,Z 745.96,A -85,B 0,C 180,E1 -17711.591,E2 -17711.591} C_VEL
LIN {X 0,Y 272.428,Z 753.961,A -85,B 0,C 180,E1 -17713.516,E2 -17713.516} C_VEL
LIN {X 0,Y 270.913,Z 761.393,A -85,B 0,C 180,E1 -17715.734,E2 -17715.734} C_VEL
LIN {X 0,Y 269.714,Z 767.361,A -85,B 0,C 180,E1 -17717.969,E2 -17717.969} C_VEL
LIN {X 0,Y 268.946,Z 772.083,A -85,B 0,C 180,E1 -17720.222,E2 -17720.222} C_VEL
LIN {X 0,Y 268.42,Z 775.695,A -85,B 0,C 180,E1 -17722.479,E2 -17722.479} C_VEL
LIN {X 0,Y 268.178,Z 778.333,A -85,B 0,C 180,E1 -17724.777,E2 -17724.777} C_VEL
LIN {X 0,Y 268.167,Z 779.953,A -85,B 0,C 180,E1 -17726.997,E2 -17726.997} C_VEL
LIN {X 0,Y 268.175,Z 780.561,A -85,B 0,C 180,E1 -17728.5,E2 -17728.5} C_VEL
LIN {X 0,Y 268.165,Z 780.821,A -85,B 0,C 180,E1 -17730.001,E2 -17730.001} C_VEL
LIN {X 0,Y 268.169,Z 782.378,A -85,B 0,C 180,E1 -17731.503,E2 -17731.503} C_VEL
LIN {X 0,Y 268.185,Z 783.37,A -85,B 0,C 180,E1 -17733.006,E2 -17733.006} C_VEL
LIN {X 0,Y 268.389,Z 783.774,A -85,B 0,C 180,E1 -17735.695,E2 -17735.695} C_VEL
LIN {X 0,Y 268.662,Z 783.111,A -85,B 0,C 180,E1 -17737.517,E2 -17737.517} C_VEL
LIN {X 0,Y 269.159,Z 782.024,A -85,B 0,C 180,E1 -17739.015,E2 -17739.015} C_VEL
LIN {X 0,Y 270.166,Z 779.262,A -85,B 0,C 180,E1 -17741.252,E2 -17741.252} C_VEL
LIN {X 0,Y 271.443,Z 775.223,A -85,B 0,C 180,E1 -17743.476,E2 -17743.476} C_VEL
LIN {X 0,Y 272.492,Z 771.798,A -85,B 0,C 180,E1 -17744.948,E2 -17744.948} C_VEL
LIN {X 0,Y 274.236,Z 766.487,A -85,B 0,C 180,E1 -17746.758,E2 -17746.758} C_VEL
LIN {X 0,Y 276.086,Z 759.945,A -85,B 0,C 180,E1 -17748.555,E2 -17748.555} C_VEL
LIN {X 0,Y 278.275,Z 751.325,A -85,B 0,C 180,E1 -17750.442,E2 -17750.442} C_VEL
LIN {X 0,Y 280.114,Z 743.125,A -85,B 0,C 180,E1 -17751.876,E2 -17751.876} C_VEL
LIN {X 0,Y 282.188,Z 733.017,A -85,B 0,C 180,E1 -17753.29,E2 -17753.29} C_VEL
LIN {X 0,Y 284.034,Z 722.122,A -85,B 0,C 180,E1 -17754.486,E2 -17754.486} C_VEL
LIN {X 0,Y 285.425,Z 712.121,A -85,B 0,C 180,E1 -17755.331,E2 -17755.331} C_VEL
LIN {X 0,Y 286.734,Z 698.631,A -85,B 0,C 180,E1 -17756.181,E2 -17756.181} C_VEL
LIN {X 0,Y 289.97,Z 668.746,A -85,B 0,C 180,E1 -17757.616,E2 -17757.616} C_VEL
LIN {X 0,Y 296.004,Z 619.885,A -85,B 0,C 180,E1 -17759.86,E2 -17759.86} C_VEL
LIN {X 0,Y 296.093,Z 616.674,A -85,B 0,C 180,E1 -17760.163,E2 -17760.163} C_VEL
LIN {X 0,Y 297.923,Z 608.662,A -85,B 0,C 180,E1 -17761.265,E2 -17761.265} C_VEL
LIN {X 0,Y 298.168,Z 605.393,A -85,B 0,C 180,E1 -17761.946,E2 -17761.946} C_VEL
LIN {X 0,Y 297.791,Z 600.222,A -85,B 0,C 180,E1 -17763.49,E2 -17763.49} C_VEL
LIN {X 0,Y 297.496,Z 598.275,A -85,B 0,C 180,E1 -17764.225,E2 -17764.225} C_VEL
LIN {X 0,Y 295.939,Z 595.37,A -85,B 0,C 180,E1 -17766.153,E2 -17766.153} C_VEL
LIN {X 0,Y 294.476,Z 593.207,A -85,B 0,C 180,E1 -17768.355,E2 -17768.355} C_VEL
LIN {X 0,Y 293.5,Z 592.21,A -85,B 0,C 180,E1 -17770.281,E2 -17770.281} C_VEL
LIN {X 0,Y 292.92,Z 591.793,A -85,B 0,C 180,E1 -17772.207,E2 -17772.207} C_VEL
LIN {X 0,Y 292.65,Z 592.015,A -85,B 0,C 180,E1 -17774.143,E2 -17774.143} C_VEL
LIN {X 0,Y 292.586,Z 592.955,A -85,B 0,C 180,E1 -17776.106,E2 -17776.106} C_VEL
LIN {X 0,Y 292.731,Z 594.631,A -85,B 0,C 180,E1 -17778.097,E2 -17778.097} C_VEL
LIN {X 0,Y 293.173,Z 597.98,A -85,B 0,C 180,E1 -17780.8,E2 -17780.8} C_VEL
LIN {X 0,Y 293.596,Z 602.219,A -85,B 0,C 180,E1 -17783.242,E2 -17783.242} C_VEL
LIN {X 0,Y 293.869,Z 607.21,A -85,B 0,C 180,E1 -17785.496,E2 -17785.496} C_VEL
LIN {X 0,Y 293.79,Z 610.204,A -85,B 0,C 180,E1 -17786.619,E2 -17786.619} C_VEL
LIN {X 0,Y 291.569,Z 618.178,A -85,B 0,C 180,E1 -17788.58,E2 -17788.58} C_VEL
LIN {X 0,Y 293.596,Z 631.258,A -85,B 0,C 180,E1 -17790.357,E2 -17790.357} C_VEL
LIN {X 0,Y 295.312,Z 644.8,A -85,B 0,C 180,E1 -17791.874,E2 -17791.874} C_VEL
LIN {X 0,Y 296.044,Z 654.436,A -85,B 0,C 180,E1 -17792.75,E2 -17792.75} C_VEL
LIN {X 0,Y 290.727,Z 702.106,A -85,B 0,C 180,E1 -17794.878,E2 -17794.878} C_VEL
LIN {X 0,Y 288.843,Z 714.314,A -85,B 0,C 180,E1 -17795.662,E2 -17795.662} C_VEL
LIN {X 0,Y 286.607,Z 725.639,A -85,B 0,C 180,E1 -17796.709,E2 -17796.709} C_VEL
LIN {X 0,Y 284.077,Z 736.659,A -85,B 0,C 180,E1 -17798.026,E2 -17798.026} C_VEL
LIN {X 0,Y 281.417,Z 746.298,A -85,B 0,C 180,E1 -17799.535,E2 -17799.535} C_VEL
LIN {X 0,Y 279.306,Z 753.308,A -85,B 0,C 180,E1 -17800.907,E2 -17800.907} C_VEL
LIN {X 0,Y 276.979,Z 760.511,A -85,B 0,C 180,E1 -17802.654,E2 -17802.654} C_VEL
LIN {X 0,Y 274.964,Z 766.345,A -85,B 0,C 180,E1 -17804.432,E2 -17804.432} C_VEL
LIN {X 0,Y 272.795,Z 771.709,A -85,B 0,C 180,E1 -17806.593,E2 -17806.593} C_VEL
LIN {X 0,Y 271.124,Z 775.666,A -85,B 0,C 180,E1 -17808.79,E2 -17808.79} C_VEL
LIN {X 0,Y 269.887,Z 778.378,A -85,B 0,C 180,E1 -17811.011,E2 -17811.011} C_VEL
LIN {X 0,Y 269.236,Z 779.571,A -85,B 0,C 180,E1 -17812.724,E2 -17812.724} C_VEL
LIN {X 0,Y 268.46,Z 780.026,A -85,B 0,C 180,E1 -17815.496,E2 -17815.496} C_VEL
LIN {X 0,Y 268.251,Z 779.576,A -85,B 0,C 180,E1 -17816.996,E2 -17816.996} C_VEL
LIN {X 0,Y 268.179,Z 778.549,A -85,B 0,C 180,E1 -17818.498,E2 -17818.498} C_VEL
LIN {X 0,Y 268.137,Z 775.918,A -85,B 0,C 180,E1 -17820.751,E2 -17820.751} C_VEL
LIN {X 0,Y 268.223,Z 773.462,A -85,B 0,C 180,E1 -17822.253,E2 -17822.253} C_VEL
LIN {X 0,Y 268.399,Z 770.326,A -85,B 0,C 180,E1 -17823.753,E2 -17823.753} C_VEL
LIN {X 0,Y 268.543,Z 764.164,A -85,B 0,C 180,E1 -17826.009,E2 -17826.009} C_VEL
LIN {X 0,Y 268.896,Z 758.303,A -85,B 0,C 180,E1 -17827.706,E2 -17827.706} C_VEL
LIN {X 0,Y 269.239,Z 751.167,A -85,B 0,C 180,E1 -17829.39,E2 -17829.39} C_VEL
LIN {X 0,Y 269.78,Z 742.276,A -85,B 0,C 180,E1 -17831.077,E2 -17831.077} C_VEL
LIN {X 0,Y 270.357,Z 733.561,A -85,B 0,C 180,E1 -17832.384,E2 -17832.384} C_VEL
LIN {X 0,Y 270.934,Z 724.382,A -85,B 0,C 180,E1 -17833.501,E2 -17833.501} C_VEL
LIN {X 0,Y 271.494,Z 713.744,A -85,B 0,C 180,E1 -17834.523,E2 -17834.523} C_VEL
LIN {X 0,Y 271.856,Z 702.052,A -85,B 0,C 180,E1 -17835.318,E2 -17835.318} C_VEL
LIN {X 0,Y 272.418,Z 688.116,A -85,B 0,C 180,E1 -17835.957,E2 -17835.957} C_VEL
LIN {X 0,Y 273.456,Z 641.742,A -85,B 0,C 180,E1 -17837.839,E2 -17837.839} C_VEL
LIN {X 0,Y 271.706,Z 618.89,A -85,B 0,C 180,E1 -17838.815,E2 -17838.815} C_VEL
LIN {X 0,Y 271.732,Z 617.016,A -85,B 0,C 180,E1 -17838.96,E2 -17838.96} C_VEL
LIN {X 0,Y 273.33,Z 596.227,A -85,B 0,C 180,E1 -17843.487,E2 -17843.487} C_VEL
LIN {X 0,Y 275.09,Z 576.466,A -85,B 0,C 180,E1 -17847.791,E2 -17847.791} C_VEL
LIN {X 0,Y 274.783,Z 572.648,A -85,B 0,C 180,E1 -17848.657,E2 -17848.657} C_VEL
LIN {X 0,Y 271.345,Z 556.081,A -85,B 0,C 180,E1 -17852.576,E2 -17852.576} C_VEL
LIN {X 0,Y 270.348,Z 550.967,A -85,B 0,C 180,E1 -17853.852,E2 -17853.852} C_VEL
LIN {X 0,Y 270.243,Z 550.823,A -85,B 0,C 180,E1 -17856.737,E2 -17856.737} C_VEL
LIN {X 0,Y 270.178,Z 550.785,A -85,B 0,C 180,E1 -17860.566,E2 -17860.566} C_VEL
LIN {X 0,Y 270.156,Z 550.802,A -85,B 0,C 180,E1 -17864.62,E2 -17864.62} C_VEL
LIN {X 0,Y 270.176,Z 550.826,A -85,B 0,C 180,E1 -17867.441,E2 -17867.441} C_VEL
LIN {X 0,Y 270.211,Z 550.792,A -85,B 0,C 180,E1 -17871.374,E2 -17871.374} C_VEL
LIN {X 0,Y 270.206,Z 550.815,A -85,B 0,C 180,E1 -17875.094,E2 -17875.094} C_VEL
LIN {X 0,Y 270.258,Z 551.039,A -85,B 0,C 180,E1 -17878.004,E2 -17878.004} C_VEL
LIN {X 0,Y 271.225,Z 555.054,A -85,B 0,C 180,E1 -17879.669,E2 -17879.669} C_VEL
LIN {X 0,Y 275.087,Z 563.329,A -85,B 0,C 180,E1 -17880.449,E2 -17880.449} C_VEL
LIN {X 0,Y 280.971,Z 576.514,A -85,B 0,C 180,E1 -17881.511,E2 -17881.511} C_VEL
LIN {X 0,Y 285.938,Z 589.684,A -85,B 0,C 180,E1 -17882.421,E2 -17882.421} C_VEL
LIN {X 0,Y 286.241,Z 592.57,A -85,B 0,C 180,E1 -17882.533,E2 -17882.533} C_VEL
LIN {X 0,Y 284.231,Z 658.383,A -85,B 0,C 180,E1 -17884.163,E2 -17884.163} C_VEL
LIN {X 0,Y 283.574,Z 670.596,A -85,B 0,C 180,E1 -17884.64,E2 -17884.64} C_VEL
LIN {X 0,Y 282.514,Z 682.878,A -85,B 0,C 180,E1 -17885.374,E2 -17885.374} C_VEL
LIN {X 0,Y 281.066,Z 695.226,A -85,B 0,C 180,E1 -17886.416,E2 -17886.416} C_VEL
LIN {X 0,Y 279.412,Z 706.309,A -85,B 0,C 180,E1 -17887.638,E2 -17887.638} C_VEL
LIN {X 0,Y 277.707,Z 716.455,A -85,B 0,C 180,E1 -17889.054,E2 -17889.054} C_VEL
LIN {X 0,Y 276.149,Z 725.764,A -85,B 0,C 180,E1 -17890.678,E2 -17890.678} C_VEL
LIN {X 0,Y 274.422,Z 734.251,A -85,B 0,C 180,E1 -17892.486,E2 -17892.486} C_VEL
LIN {X 0,Y 272.617,Z 742.499,A -85,B 0,C 180,E1 -17894.677,E2 -17894.677} C_VEL
LIN {X 0,Y 271.194,Z 749.14,A -85,B 0,C 180,E1 -17896.893,E2 -17896.893} C_VEL
LIN {X 0,Y 269.871,Z 755.225,A -85,B 0,C 180,E1 -17899.495,E2 -17899.495} C_VEL
LIN {X 0,Y 269.134,Z 759.168,A -85,B 0,C 180,E1 -17901.741,E2 -17901.741} C_VEL
LIN {X 0,Y 268.669,Z 762.078,A -85,B 0,C 180,E1 -17903.993,E2 -17903.993} C_VEL
LIN {X 0,Y 268.486,Z 763.471,A -85,B 0,C 180,E1 -17905.495,E2 -17905.495} C_VEL
LIN {X 0,Y 268.362,Z 764.463,A -85,B 0,C 180,E1 -17906.996,E2 -17906.996} C_VEL
LIN {X 0,Y 268.21,Z 765.306,A -85,B 0,C 180,E1 -17909.999,E2 -17909.999} C_VEL
LIN {X 0,Y 268.234,Z 765.114,A -85,B 0,C 180,E1 -17911.5,E2 -17911.5} C_VEL
LIN {X 0,Y 268.36,Z 764.529,A -85,B 0,C 180,E1 -17913.001,E2 -17913.001} C_VEL
LIN {X 0,Y 268.482,Z 763.564,A -85,B 0,C 180,E1 -17914.503,E2 -17914.503} C_VEL
LIN {X 0,Y 268.75,Z 761.737,A -85,B 0,C 180,E1 -17916.419,E2 -17916.419} C_VEL
LIN {X 0,Y 269.347,Z 758.145,A -85,B 0,C 180,E1 -17919.006,E2 -17919.006} C_VEL
LIN {X 0,Y 270.182,Z 753.892,A -85,B 0,C 180,E1 -17921.249,E2 -17921.249} C_VEL
LIN {X 0,Y 271.602,Z 747.453,A -85,B 0,C 180,E1 -17923.847,E2 -17923.847} C_VEL
LIN {X 0,Y 273.061,Z 740.374,A -85,B 0,C 180,E1 -17926.061,E2 -17926.061} C_VEL
LIN {X 0,Y 275.102,Z 731.547,A -85,B 0,C 180,E1 -17928.236,E2 -17928.236} C_VEL
LIN {X 0,Y 276.807,Z 722.16,A -85,B 0,C 180,E1 -17930.11,E2 -17930.11} C_VEL
LIN {X 0,Y 278.434,Z 712.466,A -85,B 0,C 180,E1 -17931.662,E2 -17931.662} C_VEL
LIN {X 0,Y 280.276,Z 701.303,A -85,B 0,C 180,E1 -17933.065,E2 -17933.065} C_VEL
LIN {X 0,Y 281.919,Z 688.76,A -85,B 0,C 180,E1 -17934.287,E2 -17934.287} C_VEL
LIN {X 0,Y 283.135,Z 676.571,A -85,B 0,C 180,E1 -17935.154,E2 -17935.154} C_VEL
LIN {X 0,Y 284.053,Z 663.037,A -85,B 0,C 180,E1 -17935.803,E2 -17935.803} C_VEL
LIN {X 0,Y 285.098,Z 632.763,A -85,B 0,C 180,E1 -17936.593,E2 -17936.593} C_VEL
LIN {X 0,Y 286.27,Z 591.106,A -85,B 0,C 180,E1 -17937.626,E2 -17937.626} C_VEL
LIN {X 0,Y 284.966,Z 586.631,A -85,B 0,C 180,E1 -17937.889,E2 -17937.889} C_VEL
LIN {X 0,Y 277.678,Z 568.756,A -85,B 0,C 180,E1 -17939.213,E2 -17939.213} C_VEL
LIN {X 0,Y 271.276,Z 555.197,A -85,B 0,C 180,E1 -17940.433,E2 -17940.433} C_VEL
LIN {X 0,Y 270.289,Z 551.314,A -85,B 0,C 180,E1 -17941.989,E2 -17941.989} C_VEL
LIN {X 0,Y 270.211,Z 550.825,A -85,B 0,C 180,E1 -17942.44,E2 -17942.44} C_VEL
LIN {X 0,Y 270.237,Z 550.816,A -85,B 0,C 180,E1 -17946.736,E2 -17946.736} C_VEL
LIN {X 0,Y 270.171,Z 550.82,A -85,B 0,C 180,E1 -17950.564,E2 -17950.564} C_VEL
LIN {X 0,Y 270.15,Z 550.814,A -85,B 0,C 180,E1 -17954.618,E2 -17954.618} C_VEL
LIN {X 0,Y 270.204,Z 550.821,A -85,B 0,C 180,E1 -17958.961,E2 -17958.961} C_VEL
LIN {X 0,Y 270.24,Z 550.793,A -85,B 0,C 180,E1 -17961.379,E2 -17961.379} C_VEL
LIN {X 0,Y 270.233,Z 550.815,A -85,B 0,C 180,E1 -17963.988,E2 -17963.988} C_VEL
LIN {X 0,Y 269.512,Z 550.915,A -85,B 0,C 180,E1 -17965.232,E2 -17965.232} C_VEL
LIN {X 0,Y 266.617,Z 551.272,A -85,B 0,C 180,E1 -17967.258,E2 -17967.258} C_VEL
LIN {X 0,Y 264.206,Z 551.571,A -85,B 0,C 180,E1 -17968.905,E2 -17968.905} C_VEL
LIN {X 0,Y 263.202,Z 551.699,A -85,B 0,C 180,E1 -17970.182,E2 -17970.182} C_VEL
LIN {X 0,Y 263.134,Z 551.7,A -85,B 0,C 180,E1 -17970.615,E2 -17970.615} C_VEL
LIN {X 0,Y 263.203,Z 551.698,A -85,B 0,C 180,E1 -17974.708,E2 -17974.708} C_VEL
LIN {X 0,Y 263.257,Z 551.689,A -85,B 0,C 180,E1 -17979.693,E2 -17979.693} C_VEL
LIN {X 0,Y 263.344,Z 551.668,A -85,B 0,C 180,E1 -17984.521,E2 -17984.521} C_VEL
LIN {X 0,Y 263.367,Z 551.665,A -85,B 0,C 180,E1 -17989.234,E2 -17989.234} C_VEL
LIN {X 0,Y 263.566,Z 551.652,A -85,B 0,C 180,E1 -17992.338,E2 -17992.338} C_VEL
LIN {X 0,Y 263.746,Z 551.625,A -85,B 0,C 180,E1 -17998.473,E2 -17998.473} C_VEL
LIN {X 0,Y 263.746,Z 551.627,A -85,B 0,C 180,E1 -18001.527,E2 -18001.527} C_VEL
LIN {X 0,Y 263.566,Z 551.652,A -85,B 0,C 180,E1 -18007.662,E2 -18007.662} C_VEL
LIN {X 0,Y 263.367,Z 551.664,A -85,B 0,C 180,E1 -18010.766,E2 -18010.766} C_VEL
LIN {X 0,Y 263.344,Z 551.669,A -85,B 0,C 180,E1 -18015.478,E2 -18015.478} C_VEL
LIN {X 0,Y 263.257,Z 551.688,A -85,B 0,C 180,E1 -18020.307,E2 -18020.307} C_VEL
LIN {X 0,Y 263.201,Z 551.697,A -85,B 0,C 180,E1 -18025.292,E2 -18025.292} C_VEL
LIN {X 0,Y 263.159,Z 551.705,A -85,B 0,C 180,E1 -18028.732,E2 -18028.732} C_VEL
LIN {X 0,Y 263.127,Z 551.708,A -85,B 0,C 180,E1 -18032.289,E2 -18032.289} C_VEL
LIN {X 0,Y 263.177,Z 551.674,A -85,B 0,C 180,E1 -18036.764,E2 -18036.764} C_VEL
LIN {X 0,Y 263.128,Z 551.71,A -85,B 0,C 180,E1 -18039.869,E2 -18039.869} C_VEL
LIN {X 0,Y 263.134,Z 551.699,A -85,B 0,C 180,E1 -18043.982,E2 -18043.982} C_VEL
LIN {X 0,Y 263.206,Z 551.695,A -85,B 0,C 180,E1 -18048.387,E2 -18048.387} C_VEL
LIN {X 0,Y 263.236,Z 551.792,A -85,B 0,C 180,E1 -18052.587,E2 -18052.587} C_VEL
LIN {X 0,Y 265.517,Z 561.596,A -85,B 0,C 180,E1 -18056.645,E2 -18056.645} C_VEL
LIN {X 0,Y 266.968,Z 568.058,A -85,B 0,C 180,E1 -18059.054,E2 -18059.054} C_VEL
LIN {X 0,Y 273.592,Z 583.715,A -85,B 0,C 180,E1 -18060.386,E2 -18060.386} C_VEL
LIN {X 0,Y 275.017,Z 587.945,A -85,B 0,C 180,E1 -18060.678,E2 -18060.678} C_VEL
LIN {X 0,Y 279.255,Z 615.002,A -85,B 0,C 180,E1 -18061.935,E2 -18061.935} C_VEL
LIN {X 0,Y 279.095,Z 624.163,A -85,B 0,C 180,E1 -18062.179,E2 -18062.179} C_VEL
LIN {X 0,Y 277.486,Z 676.545,A -85,B 0,C 180,E1 -18063.54,E2 -18063.54} C_VEL
LIN {X 0,Y 276.277,Z 690.442,A -85,B 0,C 180,E1 -18064.176,E2 -18064.176} C_VEL
LIN {X 0,Y 274.875,Z 702.89,A -85,B 0,C 180,E1 -18065.049,E2 -18065.049} C_VEL
LIN {X 0,Y 273.266,Z 714.002,A -85,B 0,C 180,E1 -18066.106,E2 -18066.106} C_VEL
LIN {X 0,Y 271.284,Z 725.571,A -85,B 0,C 180,E1 -18067.536,E2 -18067.536} C_VEL
LIN {X 0,Y 269.235,Z 735.989,A -85,B 0,C 180,E1 -18069.168,E2 -18069.168} C_VEL
LIN {X 0,Y 267.464,Z 744.867,A -85,B 0,C 180,E1 -18070.906,E2 -18070.906} C_VEL
LIN {X 0,Y 265.608,Z 753.757,A -85,B 0,C 180,E1 -18073.08,E2 -18073.08} C_VEL
LIN {X 0,Y 263.987,Z 761.188,A -85,B 0,C 180,E1 -18075.351,E2 -18075.351} C_VEL
LIN {X 0,Y 262.726,Z 767.156,A -85,B 0,C 180,E1 -18077.644,E2 -18077.644} C_VEL
LIN {X 0,Y 261.908,Z 771.878,A -85,B 0,C 180,E1 -18079.957,E2 -18079.957} C_VEL
LIN {X 0,Y 261.356,Z 775.49,A -85,B 0,C 180,E1 -18082.274,E2 -18082.274} C_VEL
LIN {X 0,Y 261.084,Z 778.348,A -85,B 0,C 180,E1 -18084.866,E2 -18084.866} C_VEL
LIN {X 0,Y 261.063,Z 779.749,A -85,B 0,C 180,E1 -18086.915,E2 -18086.915} C_VEL
LIN {X 0,Y 261.082,Z 780.357,A -85,B 0,C 180,E1 -18088.459,E2 -18088.459} C_VEL
LIN {X 0,Y 261.076,Z 780.675,A -85,B 0,C 180,E1 -18090.387,E2 -18090.387} C_VEL
LIN {X 0,Y 261.098,Z 781.904,A -85,B 0,C 180,E1 -18091.544,E2 -18091.544} C_VEL
LIN {X 0,Y 261.103,Z 783.021,A -85,B 0,C 180,E1 -18093.087,E2 -18093.087} C_VEL
LIN {X 0,Y 261.293,Z 783.806,A -85,B 0,C 180,E1 -18095.62,E2 -18095.62} C_VEL
LIN {X 0,Y 261.636,Z 783.333,A -85,B 0,C 180,E1 -18097.72,E2 -18097.72} C_VEL
LIN {X 0,Y 262.157,Z 782.327,A -85,B 0,C 180,E1 -18099.258,E2 -18099.258} C_VEL
LIN {X 0,Y 263.246,Z 779.905,A -85,B 0,C 180,E1 -18101.552,E2 -18101.552} C_VEL
LIN {X 0,Y 264.609,Z 776.18,A -85,B 0,C 180,E1 -18103.831,E2 -18103.831} C_VEL
LIN {X 0,Y 265.739,Z 773.003,A -85,B 0,C 180,E1 -18105.337,E2 -18105.337} C_VEL
LIN {X 0,Y 267.974,Z 766.797,A -85,B 0,C 180,E1 -18107.555,E2 -18107.555} C_VEL
LIN {X 0,Y 270.02,Z 760.423,A -85,B 0,C 180,E1 -18109.383,E2 -18109.383} C_VEL
LIN {X 0,Y 272.283,Z 752.587,A -85,B 0,C 180,E1 -18111.185,E2 -18111.185} C_VEL
LIN {X 0,Y 274.231,Z 744.895,A -85,B 0,C 180,E1 -18112.609,E2 -18112.609} C_VEL
LIN {X 0,Y 276.402,Z 735.571,A -85,B 0,C 180,E1 -18114.007,E2 -18114.007} C_VEL
LIN {X 0,Y 278.449,Z 725.503,A -85,B 0,C 180,E1 -18115.21,E2 -18115.21} C_VEL
LIN {X 0,Y 280.415,Z 713.349,A -85,B 0,C 180,E1 -18116.316,E2 -18116.316} C_VEL
LIN {X 0,Y 281.915,Z 700.864,A -85,B 0,C 180,E1 -18117.164,E2 -18117.164} C_VEL
LIN {X 0,Y 285.146,Z 672.368,A -85,B 0,C 180,E1 -18118.576,E2 -18118.576} C_VEL
LIN {X 0,Y 291.959,Z 621.505,A -85,B 0,C 180,E1 -18120.954,E2 -18120.954} C_VEL
LIN {X 0,Y 292.025,Z 616.977,A -85,B 0,C 180,E1 -18121.389,E2 -18121.389} C_VEL
LIN {X 0,Y 293.265,Z 612.175,A -85,B 0,C 180,E1 -18122.061,E2 -18122.061} C_VEL
LIN {X 0,Y 293.576,Z 609.436,A -85,B 0,C 180,E1 -18122.646,E2 -18122.646} C_VEL
LIN {X 0,Y 293.286,Z 604.879,A -85,B 0,C 180,E1 -18124.075,E2 -18124.075} C_VEL
LIN {X 0,Y 293.089,Z 603.584,A -85,B 0,C 180,E1 -18124.586,E2 -18124.586} C_VEL
LIN {X 0,Y 291.987,Z 601.445,A -85,B 0,C 180,E1 -18125.976,E2 -18125.976} C_VEL
LIN {X 0,Y 291.087,Z 600.063,A -85,B 0,C 180,E1 -18127.179,E2 -18127.179} C_VEL
LIN {X 0,Y 289.887,Z 598.519,A -85,B 0,C 180,E1 -18129.122,E2 -18129.122} C_VEL
LIN {X 0,Y 288.98,Z 597.724,A -85,B 0,C 180,E1 -18131.069,E2 -18131.069} C_VEL
LIN {X 0,Y 288.465,Z 597.519,A -85,B 0,C 180,E1 -18133.038,E2 -18133.038} C_VEL
LIN {X 0,Y 288.191,Z 597.992,A -85,B 0,C 180,E1 -18135.01,E2 -18135.01} C_VEL
LIN {X 0,Y 288.131,Z 599.234,A -85,B 0,C 180,E1 -18137.035,E2 -18137.035} C_VEL
LIN {X 0,Y 288.356,Z 602.578,A -85,B 0,C 180,E1 -18140.17,E2 -18140.17} C_VEL
LIN {X 0,Y 288.572,Z 606.264,A -85,B 0,C 180,E1 -18142.493,E2 -18142.493} C_VEL
LIN {X 0,Y 288.749,Z 610.527,A -85,B 0,C 180,E1 -18144.615,E2 -18144.615} C_VEL
LIN {X 0,Y 288.642,Z 613.824,A -85,B 0,C 180,E1 -18145.943,E2 -18145.943} C_VEL
LIN {X 0,Y 287.349,Z 618.247,A -85,B 0,C 180,E1 -18147.069,E2 -18147.069} C_VEL
LIN {X 0,Y 289.265,Z 632.563,A -85,B 0,C 180,E1 -18149.154,E2 -18149.154} C_VEL
LIN {X 0,Y 290.701,Z 645.185,A -85,B 0,C 180,E1 -18150.675,E2 -18150.675} C_VEL
LIN {X 0,Y 291.444,Z 655.421,A -85,B 0,C 180,E1 -18151.7,E2 -18151.7} C_VEL
LIN {X 0,Y 285.876,Z 701.975,A -85,B 0,C 180,E1 -18153.834,E2 -18153.834} C_VEL
LIN {X 0,Y 283.868,Z 714.036,A -85,B 0,C 180,E1 -18154.62,E2 -18154.62} C_VEL
LIN {X 0,Y 281.514,Z 725.476,A -85,B 0,C 180,E1 -18155.674,E2 -18155.674} C_VEL
LIN {X 0,Y 279.429,Z 733.934,A -85,B 0,C 180,E1 -18156.663,E2 -18156.663} C_VEL
LIN {X 0,Y 276.863,Z 743.185,A -85,B 0,C 180,E1 -18158.012,E2 -18158.012} C_VEL
LIN {X 0,Y 273.91,Z 752.298,A -85,B 0,C 180,E1 -18159.734,E2 -18159.734} C_VEL
LIN {X 0,Y 271.818,Z 758.341,A -85,B 0,C 180,E1 -18161.144,E2 -18161.144} C_VEL
LIN {X 0,Y 269.482,Z 764.554,A -85,B 0,C 180,E1 -18162.939,E2 -18162.939} C_VEL
LIN {X 0,Y 267.49,Z 769.531,A -85,B 0,C 180,E1 -18164.767,E2 -18164.767} C_VEL
LIN {X 0,Y 265.354,Z 774.164,A -85,B 0,C 180,E1 -18166.99,E2 -18166.99} C_VEL
LIN {X 0,Y 263.714,Z 777.342,A -85,B 0,C 180,E1 -18169.248,E2 -18169.248} C_VEL
LIN {X 0,Y 262.886,Z 778.836,A -85,B 0,C 180,E1 -18170.77,E2 -18170.77} C_VEL
LIN {X 0,Y 262.086,Z 779.938,A -85,B 0,C 180,E1 -18172.835,E2 -18172.835} C_VEL
LIN {X 0,Y 261.384,Z 779.99,A -85,B 0,C 180,E1 -18175.373,E2 -18175.373} C_VEL
LIN {X 0,Y 261.174,Z 779.345,A -85,B 0,C 180,E1 -18176.915,E2 -18176.915} C_VEL
LIN {X 0,Y 261.11,Z 778.193,A -85,B 0,C 180,E1 -18178.458,E2 -18178.458} C_VEL
LIN {X 0,Y 261.067,Z 775.315,A -85,B 0,C 180,E1 -18180.771,E2 -18180.771} C_VEL
LIN {X 0,Y 261.26,Z 771.122,A -85,B 0,C 180,E1 -18183.084,E2 -18183.084} C_VEL
LIN {X 0,Y 261.371,Z 765.962,A -85,B 0,C 180,E1 -18185.183,E2 -18185.183} C_VEL
LIN {X 0,Y 261.794,Z 758.994,A -85,B 0,C 180,E1 -18187.326,E2 -18187.326} C_VEL
LIN {X 0,Y 262.05,Z 752.775,A -85,B 0,C 180,E1 -18188.871,E2 -18188.871} C_VEL
LIN {X 0,Y 262.57,Z 744.301,A -85,B 0,C 180,E1 -18190.604,E2 -18190.604} C_VEL
LIN {X 0,Y 263.195,Z 734.827,A -85,B 0,C 180,E1 -18192.139,E2 -18192.139} C_VEL
LIN {X 0,Y 263.724,Z 725.946,A -85,B 0,C 180,E1 -18193.288,E2 -18193.288} C_VEL
LIN {X 0,Y 264.313,Z 715.792,A -85,B 0,C 180,E1 -18194.337,E2 -18194.337} C_VEL
LIN {X 0,Y 264.681,Z 703.783,A -85,B 0,C 180,E1 -18195.251,E2 -18195.251} C_VEL
LIN {X 0,Y 265.245,Z 690.844,A -85,B 0,C 180,E1 -18195.907,E2 -18195.907} C_VEL
LIN {X 0,Y 266.407,Z 642.311,A -85,B 0,C 180,E1 -18197.944,E2 -18197.944} C_VEL
LIN {X 0,Y 264.695,Z 620.012,A -85,B 0,C 180,E1 -18198.931,E2 -18198.931} C_VEL
LIN {X 0,Y 264.661,Z 617.254,A -85,B 0,C 180,E1 -18199.084,E2 -18199.084} C_VEL
LIN {X 0,Y 266.334,Z 596.298,A -85,B 0,C 180,E1 -18203.729,E2 -18203.729} C_VEL
LIN {X 0,Y 267.992,Z 578.146,A -85,B 0,C 180,E1 -18207.754,E2 -18207.754} C_VEL
LIN {X 0,Y 267.901,Z 574.407,A -85,B 0,C 180,E1 -18208.605,E2 -18208.605} C_VEL
LIN {X 0,Y 264.484,Z 557.959,A -85,B 0,C 180,E1 -18212.554,E2 -18212.554} C_VEL
LIN {X 0,Y 263.295,Z 551.825,A -85,B 0,C 180,E1 -18214.121,E2 -18214.121} C_VEL
LIN {X 0,Y 263.17,Z 551.702,A -85,B 0,C 180,E1 -18217.895,E2 -18217.895} C_VEL
LIN {X 0,Y 263.127,Z 551.649,A -85,B 0,C 180,E1 -18221.893,E2 -18221.893} C_VEL
LIN {X 0,Y 263.128,Z 551.708,A -85,B 0,C 180,E1 -18226.15,E2 -18226.15} C_VEL
LIN {X 0,Y 263.109,Z 551.67,A -85,B 0,C 180,E1 -18230.127,E2 -18230.127} C_VEL
LIN {X 0,Y 263.167,Z 551.701,A -85,B 0,C 180,E1 -18234.017,E2 -18234.017} C_VEL
LIN {X 0,Y 263.182,Z 551.851,A -85,B 0,C 180,E1 -18237.264,E2 -18237.264} C_VEL
LIN {X 0,Y 264.028,Z 555.237,A -85,B 0,C 180,E1 -18238.738,E2 -18238.738} C_VEL
LIN {X 0,Y 266.263,Z 560.026,A -85,B 0,C 180,E1 -18239.255,E2 -18239.255} C_VEL
LIN {X 0,Y 273.83,Z 576.269,A -85,B 0,C 180,E1 -18240.682,E2 -18240.682} C_VEL
LIN {X 0,Y 279.846,Z 591.786,A -85,B 0,C 180,E1 -18241.822,E2 -18241.822} C_VEL
LIN {X 0,Y 278.047,Z 655.534,A -85,B 0,C 180,E1 -18243.443,E2 -18243.443} C_VEL
LIN {X 0,Y 277.338,Z 668.072,A -85,B 0,C 180,E1 -18243.876,E2 -18243.876} C_VEL
LIN {X 0,Y 276.367,Z 680.506,A -85,B 0,C 180,E1 -18244.586,E2 -18244.586} C_VEL
LIN {X 0,Y 275.101,Z 691.692,A -85,B 0,C 180,E1 -18245.471,E2 -18245.471} C_VEL
LIN {X 0,Y 273.338,Z 703.66,A -85,B 0,C 180,E1 -18246.713,E2 -18246.713} C_VEL
LIN {X 0,Y 271.516,Z 714.323,A -85,B 0,C 180,E1 -18248.154,E2 -18248.154} C_VEL
LIN {X 0,Y 269.67,Z 724.773,A -85,B 0,C 180,E1 -18249.95,E2 -18249.95} C_VEL
LIN {X 0,Y 267.658,Z 734.458,A -85,B 0,C 180,E1 -18252.028,E2 -18252.028} C_VEL
LIN {X 0,Y 265.783,Z 742.706,A -85,B 0,C 180,E1 -18254.273,E2 -18254.273} C_VEL
